LIN {X 0,Y 525.083,Z 545.384,A -85,B 0,C 180,E1 -4788.258,E2 -4788.258} C_VEL
LIN {X 0,Y 525.597,Z 520.306,A -85,B 0,C 180,E1 -4791.163,E2 -4791.163} C_VEL
LIN {X 0,Y 526.091,Z 495.739,A -85,B 0,C 180,E1 -4794.044,E2 -4794.044} C_VEL
LIN {X 0,Y 526.597,Z 472.119,A -85,B 0,C 180,E1 -4796.856,E2 -4796.856} C_VEL
LIN {X 0,Y 524.984,Z 463.792,A -85,B 0,C 180,E1 -4797.939,E2 -4797.939} C_VEL
LIN {X 0,Y 524.003,Z 459.339,A -85,B 0,C 180,E1 -4798.569,E2 -4798.569} C_VEL
LIN {X 0,Y 523.92,Z 459.219,A -85,B 0,C 180,E1 -4801.543,E2 -4801.543} C_VEL
LIN {X 0,Y 523.931,Z 459.225,A -85,B 0,C 180,E1 -4804.289,E2 -4804.289} C_VEL
LIN {X 0,Y 523.905,Z 459.219,A -85,B 0,C 180,E1 -4807.131,E2 -4807.131} C_VEL
LIN {X 0,Y 523.965,Z 459.214,A -85,B 0,C 180,E1 -4810.133,E2 -4810.133} C_VEL
LIN {X 0,Y 523.921,Z 459.219,A -85,B 0,C 180,E1 -4813.166,E2 -4813.166} C_VEL
LIN {X 0,Y 523.936,Z 459.213,A -85,B 0,C 180,E1 -4815.771,E2 -4815.771} C_VEL
LIN {X 0,Y 523.939,Z 459.217,A -85,B 0,C 180,E1 -4818.907,E2 -4818.907} C_VEL
LIN {X 0,Y 523.911,Z 459.221,A -85,B 0,C 180,E1 -4821.898,E2 -4821.898} C_VEL
LIN {X 0,Y 523.933,Z 459.217,A -85,B 0,C 180,E1 -4824.908,E2 -4824.908} C_VEL
LIN {X 0,Y 523.936,Z 459.214,A -85,B 0,C 180,E1 -4827.677,E2 -4827.677} C_VEL
LIN {X 0,Y 523.962,Z 459.216,A -85,B 0,C 180,E1 -4830.673,E2 -4830.673} C_VEL
LIN {X 0,Y 523.97,Z 459.207,A -85,B 0,C 180,E1 -4833.728,E2 -4833.728} C_VEL
LIN {X 0,Y 523.928,Z 459.224,A -85,B 0,C 180,E1 -4836.27,E2 -4836.27} C_VEL
LIN {X 0,Y 523.938,Z 459.216,A -85,B 0,C 180,E1 -4838.766,E2 -4838.766} C_VEL
LIN {X 0,Y 523.945,Z 459.207,A -85,B 0,C 180,E1 -4841.22,E2 -4841.22} C_VEL
LIN {X 0,Y 523.931,Z 459.215,A -85,B 0,C 180,E1 -4843.639,E2 -4843.639} C_VEL
LIN {X 0,Y 523.931,Z 459.22,A -85,B 0,C 180,E1 -4846.028,E2 -4846.028} C_VEL
LIN {X 0,Y 524.002,Z 459.213,A -85,B 0,C 180,E1 -4848.394,E2 -4848.394} C_VEL
LIN {X 0,Y 523.999,Z 459.208,A -85,B 0,C 180,E1 -4851.516,E2 -4851.516} C_VEL
LIN {X 0,Y 524.09,Z 459.2,A -85,B 0,C 180,E1 -4854.614,E2 -4854.614} C_VEL
LIN {X 0,Y 524.103,Z 459.194,A -85,B 0,C 180,E1 -4857.694,E2 -4857.694} C_VEL
LIN {X 0,Y 524.117,Z 459.197,A -85,B 0,C 180,E1 -4860.768,E2 -4860.768} C_VEL
LIN {X 0,Y 524.067,Z 459.199,A -85,B 0,C 180,E1 -4863.075,E2 -4863.075} C_VEL
LIN {X 0,Y 524.042,Z 459.205,A -85,B 0,C 180,E1 -4866.159,E2 -4866.159} C_VEL
LIN {X 0,Y 523.995,Z 459.205,A -85,B 0,C 180,E1 -4869.262,E2 -4869.262} C_VEL
LIN {X 0,Y 523.998,Z 459.207,A -85,B 0,C 180,E1 -4871.743,E2 -4871.743} C_VEL
LIN {X 0,Y 523.984,Z 459.21,A -85,B 0,C 180,E1 -4875.053,E2 -4875.053} C_VEL
LIN {X 0,Y 523.955,Z 459.213,A -85,B 0,C 180,E1 -4877.969,E2 -4877.969} C_VEL
LIN {X 0,Y 523.964,Z 459.217,A -85,B 0,C 180,E1 -4880.41,E2 -4880.41} C_VEL
LIN {X 0,Y 523.909,Z 459.225,A -85,B 0,C 180,E1 -4882.894,E2 -4882.894} C_VEL
LIN {X 0,Y 523.947,Z 459.216,A -85,B 0,C 180,E1 -4885.419,E2 -4885.419} C_VEL
LIN {X 0,Y 523.963,Z 459.21,A -85,B 0,C 180,E1 -4887.999,E2 -4887.999} C_VEL
LIN {X 0,Y 523.945,Z 459.209,A -85,B 0,C 180,E1 -4890.857,E2 -4890.857} C_VEL
LIN {X 0,Y 523.957,Z 459.212,A -85,B 0,C 180,E1 -4893.736,E2 -4893.736} C_VEL
LIN {X 0,Y 523.917,Z 459.221,A -85,B 0,C 180,E1 -4896.405,E2 -4896.405} C_VEL
LIN {X 0,Y 523.918,Z 459.214,A -85,B 0,C 180,E1 -4899.085,E2 -4899.085} C_VEL
LIN {X 0,Y 523.952,Z 459.211,A -85,B 0,C 180,E1 -4902.119,E2 -4902.119} C_VEL
LIN {X 0,Y 523.953,Z 459.216,A -85,B 0,C 180,E1 -4905.309,E2 -4905.309} C_VEL
LIN {X 0,Y 523.92,Z 459.219,A -85,B 0,C 180,E1 -4906.928,E2 -4906.928} C_VEL
LIN {X 0,Y 523.253,Z 459.298,A -85,B 0,C 180,E1 -4907.569,E2 -4907.569} C_VEL
LIN {X 0,Y 520.407,Z 459.654,A -85,B 0,C 180,E1 -4908.611,E2 -4908.611} C_VEL
LIN {X 0,Y 518.001,Z 459.959,A -85,B 0,C 180,E1 -4909.45,E2 -4909.45} C_VEL
LIN {X 0,Y 516.965,Z 460.085,A -85,B 0,C 180,E1 -4910.098,E2 -4910.098} C_VEL
LIN {X 0,Y 516.879,Z 460.096,A -85,B 0,C 180,E1 -4910.317,E2 -4910.317} C_VEL
LIN {X 0,Y 516.882,Z 460.088,A -85,B 0,C 180,E1 -4913.343,E2 -4913.343} C_VEL
LIN {X 0,Y 516.91,Z 460.075,A -85,B 0,C 180,E1 -4916.122,E2 -4916.122} C_VEL
LIN {X 0,Y 516.892,Z 460.099,A -85,B 0,C 180,E1 -4918.936,E2 -4918.936} C_VEL
LIN {X 0,Y 516.919,Z 460.086,A -85,B 0,C 180,E1 -4921.586,E2 -4921.586} C_VEL
LIN {X 0,Y 516.932,Z 460.086,A -85,B 0,C 180,E1 -4924.212,E2 -4924.212} C_VEL
LIN {X 0,Y 516.867,Z 460.102,A -85,B 0,C 180,E1 -4926.777,E2 -4926.777} C_VEL
LIN {X 0,Y 516.942,Z 460.091,A -85,B 0,C 180,E1 -4929.732,E2 -4929.732} C_VEL
LIN {X 0,Y 516.922,Z 460.066,A -85,B 0,C 180,E1 -4932.596,E2 -4932.596} C_VEL
LIN {X 0,Y 516.972,Z 460.252,A -85,B 0,C 180,E1 -4934.934,E2 -4934.934} C_VEL
LIN {X 0,Y 517.22,Z 461.336,A -85,B 0,C 180,E1 -4935.069,E2 -4935.069} C_VEL
LIN {X 0,Y 519.188,Z 467.428,A -85,B 0,C 180,E1 -4935.228,E2 -4935.228} C_VEL
LIN {X 0,Y 518.873,Z 540.381,A -85,B 0,C 180,E1 -4936.264,E2 -4936.264} C_VEL
LIN {X 0,Y 518.787,Z 553.491,A -85,B 0,C 180,E1 -4936.611,E2 -4936.611} C_VEL
LIN {X 0,Y 518.611,Z 565.176,A -85,B 0,C 180,E1 -4937.065,E2 -4937.065} C_VEL
LIN {X 0,Y 518.456,Z 576.909,A -85,B 0,C 180,E1 -4937.679,E2 -4937.679} C_VEL
LIN {X 0,Y 518.112,Z 588.391,A -85,B 0,C 180,E1 -4938.459,E2 -4938.459} C_VEL
LIN {X 0,Y 517.82,Z 598.74,A -85,B 0,C 180,E1 -4939.344,E2 -4939.344} C_VEL
LIN {X 0,Y 517.541,Z 607.185,A -85,B 0,C 180,E1 -4940.227,E2 -4940.227} C_VEL
LIN {X 0,Y 517.36,Z 614.938,A -85,B 0,C 180,E1 -4941.21,E2 -4941.21} C_VEL
LIN {X 0,Y 517.085,Z 622.633,A -85,B 0,C 180,E1 -4942.405,E2 -4942.405} C_VEL
LIN {X 0,Y 516.937,Z 629.45,A -85,B 0,C 180,E1 -4943.756,E2 -4943.756} C_VEL
LIN {X 0,Y 516.696,Z 634.082,A -85,B 0,C 180,E1 -4944.928,E2 -4944.928} C_VEL
LIN {X 0,Y 516.651,Z 637.608,A -85,B 0,C 180,E1 -4946.1,E2 -4946.1} C_VEL
LIN {X 0,Y 516.59,Z 639.435,A -85,B 0,C 180,E1 -4946.881,E2 -4946.881} C_VEL
LIN {X 0,Y 516.577,Z 640.809,A -85,B 0,C 180,E1 -4947.661,E2 -4947.661} C_VEL
LIN {X 0,Y 516.545,Z 642.388,A -85,B 0,C 180,E1 -4949.22,E2 -4949.22} C_VEL
LIN {X 0,Y 516.533,Z 642.622,A -85,B 0,C 180,E1 -4950,E2 -4950} C_VEL
LIN {X 0,Y 516.544,Z 642.442,A -85,B 0,C 180,E1 -4950.78,E2 -4950.78} C_VEL
LIN {X 0,Y 516.577,Z 640.931,A -85,B 0,C 180,E1 -4952.339,E2 -4952.339} C_VEL
LIN {X 0,Y 516.588,Z 639.612,A -85,B 0,C 180,E1 -4953.119,E2 -4953.119} C_VEL
LIN {X 0,Y 516.707,Z 636.807,A -85,B 0,C 180,E1 -4954.29,E2 -4954.29} C_VEL
LIN {X 0,Y 516.814,Z 633.006,A -85,B 0,C 180,E1 -4955.462,E2 -4955.462} C_VEL
LIN {X 0,Y 516.897,Z 627.894,A -85,B 0,C 180,E1 -4956.683,E2 -4956.683} C_VEL
LIN {X 0,Y 517.088,Z 621.918,A -85,B 0,C 180,E1 -4957.811,E2 -4957.811} C_VEL
LIN {X 0,Y 517.386,Z 614.15,A -85,B 0,C 180,E1 -4958.987,E2 -4958.987} C_VEL
LIN {X 0,Y 517.646,Z 604.487,A -85,B 0,C 180,E1 -4960.166,E2 -4960.166} C_VEL
LIN {X 0,Y 517.964,Z 595.465,A -85,B 0,C 180,E1 -4961.049,E2 -4961.049} C_VEL
LIN {X 0,Y 518.262,Z 584.994,A -85,B 0,C 180,E1 -4961.88,E2 -4961.88} C_VEL
LIN {X 0,Y 518.475,Z 573.353,A -85,B 0,C 180,E1 -4962.615,E2 -4962.615} C_VEL
LIN {X 0,Y 518.637,Z 561.959,A -85,B 0,C 180,E1 -4963.169,E2 -4963.169} C_VEL
LIN {X 0,Y 518.811,Z 549.167,A -85,B 0,C 180,E1 -4963.613,E2 -4963.613} C_VEL
LIN {X 0,Y 518.869,Z 537.032,A -85,B 0,C 180,E1 -4963.886,E2 -4963.886} C_VEL
LIN {X 0,Y 519.114,Z 466.662,A -85,B 0,C 180,E1 -4964.875,E2 -4964.875} C_VEL
LIN {X 0,Y 517.159,Z 461.11,A -85,B 0,C 180,E1 -4965.032,E2 -4965.032} C_VEL
LIN {X 0,Y 516.968,Z 460.206,A -85,B 0,C 180,E1 -4965.174,E2 -4965.174} C_VEL
LIN {X 0,Y 516.928,Z 460.073,A -85,B 0,C 180,E1 -4968.222,E2 -4968.222} C_VEL
LIN {X 0,Y 516.915,Z 460.099,A -85,B 0,C 180,E1 -4970.701,E2 -4970.701} C_VEL
LIN {X 0,Y 516.904,Z 460.093,A -85,B 0,C 180,E1 -4974.072,E2 -4974.072} C_VEL
LIN {X 0,Y 516.925,Z 460.087,A -85,B 0,C 180,E1 -4976.657,E2 -4976.657} C_VEL
LIN {X 0,Y 516.911,Z 460.094,A -85,B 0,C 180,E1 -4979.523,E2 -4979.523} C_VEL
LIN {X 0,Y 516.9,Z 460.093,A -85,B 0,C 180,E1 -4982.543,E2 -4982.543} C_VEL
LIN {X 0,Y 516.877,Z 460.098,A -85,B 0,C 180,E1 -4985.331,E2 -4985.331} C_VEL
LIN {X 0,Y 516.88,Z 460.094,A -85,B 0,C 180,E1 -4987.942,E2 -4987.942} C_VEL
LIN {X 0,Y 516.883,Z 460.1,A -85,B 0,C 180,E1 -4990.741,E2 -4990.741} C_VEL
LIN {X 0,Y 516.902,Z 460.092,A -85,B 0,C 180,E1 -4992.828,E2 -4992.828} C_VEL
LIN {X 0,Y 516.919,Z 460.096,A -85,B 0,C 180,E1 -4995.009,E2 -4995.009} C_VEL
LIN {X 0,Y 516.912,Z 460.089,A -85,B 0,C 180,E1 -4998.397,E2 -4998.397} C_VEL
LIN {X 0,Y 516.877,Z 460.096,A -85,B 0,C 180,E1 -5001.284,E2 -5001.284} C_VEL
LIN {X 0,Y 516.885,Z 460.095,A -85,B 0,C 180,E1 -5004.221,E2 -5004.221} C_VEL
LIN {X 0,Y 516.892,Z 460.097,A -85,B 0,C 180,E1 -5007.053,E2 -5007.053} C_VEL
LIN {X 0,Y 516.895,Z 460.083,A -85,B 0,C 180,E1 -5009.796,E2 -5009.796} C_VEL
LIN {X 0,Y 516.923,Z 460.087,A -85,B 0,C 180,E1 -5012.467,E2 -5012.467} C_VEL
LIN {X 0,Y 516.904,Z 460.099,A -85,B 0,C 180,E1 -5015.071,E2 -5015.071} C_VEL
LIN {X 0,Y 516.878,Z 460.092,A -85,B 0,C 180,E1 -5018.462,E2 -5018.462} C_VEL
LIN {X 0,Y 516.896,Z 460.097,A -85,B 0,C 180,E1 -5020.955,E2 -5020.955} C_VEL
LIN {X 0,Y 516.908,Z 460.095,A -85,B 0,C 180,E1 -5023.41,E2 -5023.41} C_VEL
LIN {X 0,Y 516.896,Z 460.095,A -85,B 0,C 180,E1 -5025.834,E2 -5025.834} C_VEL
LIN {X 0,Y 516.948,Z 460.09,A -85,B 0,C 180,E1 -5029.028,E2 -5029.028} C_VEL
LIN {X 0,Y 516.969,Z 460.082,A -85,B 0,C 180,E1 -5032.187,E2 -5032.187} C_VEL
LIN {X 0,Y 517.023,Z 460.076,A -85,B 0,C 180,E1 -5034.54,E2 -5034.54} C_VEL
LIN {X 0,Y 517.075,Z 460.073,A -85,B 0,C 180,E1 -5037.663,E2 -5037.663} C_VEL
LIN {X 0,Y 517.086,Z 460.069,A -85,B 0,C 180,E1 -5040.779,E2 -5040.779} C_VEL
LIN {X 0,Y 517.008,Z 460.081,A -85,B 0,C 180,E1 -5043.117,E2 -5043.117} C_VEL
LIN {X 0,Y 517.001,Z 460.08,A -85,B 0,C 180,E1 -5046.243,E2 -5046.243} C_VEL
LIN {X 0,Y 516.948,Z 460.093,A -85,B 0,C 180,E1 -5049.389,E2 -5049.389} C_VEL
LIN {X 0,Y 516.947,Z 460.09,A -85,B 0,C 180,E1 -5051.81,E2 -5051.81} C_VEL
LIN {X 0,Y 516.934,Z 460.092,A -85,B 0,C 180,E1 -5055.147,E2 -5055.147} C_VEL
LIN {X 0,Y 516.917,Z 460.082,A -85,B 0,C 180,E1 -5058.223,E2 -5058.223} C_VEL
LIN {X 0,Y 516.904,Z 460.088,A -85,B 0,C 180,E1 -5060.702,E2 -5060.702} C_VEL
LIN {X 0,Y 516.903,Z 460.094,A -85,B 0,C 180,E1 -5064.072,E2 -5064.072} C_VEL
LIN {X 0,Y 516.921,Z 460.083,A -85,B 0,C 180,E1 -5066.658,E2 -5066.658} C_VEL
LIN {X 0,Y 516.917,Z 460.096,A -85,B 0,C 180,E1 -5069.527,E2 -5069.527} C_VEL
LIN {X 0,Y 516.894,Z 460.089,A -85,B 0,C 180,E1 -5072.545,E2 -5072.545} C_VEL
LIN {X 0,Y 516.877,Z 460.098,A -85,B 0,C 180,E1 -5075.333,E2 -5075.333} C_VEL
LIN {X 0,Y 516.875,Z 460.099,A -85,B 0,C 180,E1 -5077.944,E2 -5077.944} C_VEL
LIN {X 0,Y 516.88,Z 460.096,A -85,B 0,C 180,E1 -5080.742,E2 -5080.742} C_VEL
LIN {X 0,Y 516.879,Z 460.09,A -85,B 0,C 180,E1 -5082.832,E2 -5082.832} C_VEL
LIN {X 0,Y 516.918,Z 460.085,A -85,B 0,C 180,E1 -5085.011,E2 -5085.011} C_VEL
LIN {X 0,Y 516.919,Z 460.089,A -85,B 0,C 180,E1 -5088.398,E2 -5088.398} C_VEL
LIN {X 0,Y 516.884,Z 460.097,A -85,B 0,C 180,E1 -5091.285,E2 -5091.285} C_VEL
LIN {X 0,Y 516.885,Z 460.1,A -85,B 0,C 180,E1 -5094.222,E2 -5094.222} C_VEL
LIN {X 0,Y 516.895,Z 460.093,A -85,B 0,C 180,E1 -5097.054,E2 -5097.054} C_VEL
LIN {X 0,Y 516.892,Z 460.082,A -85,B 0,C 180,E1 -5099.797,E2 -5099.797} C_VEL
LIN {X 0,Y 516.955,Z 460.3,A -85,B 0,C 180,E1 -5101.255,E2 -5101.255} C_VEL
LIN {X 0,Y 519.648,Z 472.95,A -85,B 0,C 180,E1 -5102.969,E2 -5102.969} C_VEL
LIN {X 0,Y 519.241,Z 493.076,A -85,B 0,C 180,E1 -5105.405,E2 -5105.405} C_VEL
LIN {X 0,Y 518.715,Z 515.897,A -85,B 0,C 180,E1 -5108.125,E2 -5108.125} C_VEL
LIN {X 0,Y 518.097,Z 544.156,A -85,B 0,C 180,E1 -5111.452,E2 -5111.452} C_VEL
LIN {X 0,Y 517.588,Z 571.268,A -85,B 0,C 180,E1 -5114.594,E2 -5114.594} C_VEL
LIN {X 0,Y 519.083,Z 584.74,A -85,B 0,C 180,E1 -5114.848,E2 -5114.848} C_VEL
LIN {X 0,Y 518.599,Z 681.826,A -85,B 0,C 180,E1 -5116.207,E2 -5116.207} C_VEL
LIN {X 0,Y 518.313,Z 695.176,A -85,B 0,C 180,E1 -5116.548,E2 -5116.548} C_VEL
LIN {X 0,Y 518.074,Z 708.587,A -85,B 0,C 180,E1 -5117.066,E2 -5117.066} C_VEL
LIN {X 0,Y 517.77,Z 720.716,A -85,B 0,C 180,E1 -5117.709,E2 -5117.709} C_VEL
LIN {X 0,Y 517.459,Z 732.937,A -85,B 0,C 180,E1 -5118.543,E2 -5118.543} C_VEL
LIN {X 0,Y 517.153,Z 743.295,A -85,B 0,C 180,E1 -5119.429,E2 -5119.429} C_VEL
LIN {X 0,Y 516.925,Z 752.639,A -85,B 0,C 180,E1 -5120.413,E2 -5120.413} C_VEL
LIN {X 0,Y 516.686,Z 761.755,A -85,B 0,C 180,E1 -5121.592,E2 -5121.592} C_VEL
LIN {X 0,Y 516.51,Z 769.109,A -85,B 0,C 180,E1 -5122.77,E2 -5122.77} C_VEL
LIN {X 0,Y 516.454,Z 775.831,A -85,B 0,C 180,E1 -5124.142,E2 -5124.142} C_VEL
LIN {X 0,Y 516.271,Z 780.26,A -85,B 0,C 180,E1 -5125.315,E2 -5125.315} C_VEL
LIN {X 0,Y 516.372,Z 782.633,A -85,B 0,C 180,E1 -5126.098,E2 -5126.098} C_VEL
LIN {X 0,Y 516.282,Z 784.534,A -85,B 0,C 180,E1 -5126.879,E2 -5126.879} C_VEL
LIN {X 0,Y 516.26,Z 785.967,A -85,B 0,C 180,E1 -5127.659,E2 -5127.659} C_VEL
LIN {X 0,Y 516.16,Z 787.598,A -85,B 0,C 180,E1 -5129.22,E2 -5129.22} C_VEL
LIN {X 0,Y 516.154,Z 787.819,A -85,B 0,C 180,E1 -5130,E2 -5130} C_VEL
LIN {X 0,Y 516.16,Z 787.599,A -85,B 0,C 180,E1 -5130.78,E2 -5130.78} C_VEL
LIN {X 0,Y 516.26,Z 785.97,A -85,B 0,C 180,E1 -5132.341,E2 -5132.341} C_VEL
LIN {X 0,Y 516.282,Z 784.538,A -85,B 0,C 180,E1 -5133.121,E2 -5133.121} C_VEL
LIN {X 0,Y 516.326,Z 781.528,A -85,B 0,C 180,E1 -5134.293,E2 -5134.293} C_VEL
LIN {X 0,Y 516.405,Z 777.459,A -85,B 0,C 180,E1 -5135.467,E2 -5135.467} C_VEL
LIN {X 0,Y 516.465,Z 772.035,A -85,B 0,C 180,E1 -5136.678,E2 -5136.678} C_VEL
LIN {X 0,Y 516.578,Z 765.631,A -85,B 0,C 180,E1 -5137.819,E2 -5137.819} C_VEL
LIN {X 0,Y 516.787,Z 757.439,A -85,B 0,C 180,E1 -5138.997,E2 -5138.997} C_VEL
LIN {X 0,Y 517.02,Z 749.107,A -85,B 0,C 180,E1 -5139.98,E2 -5139.98} C_VEL
LIN {X 0,Y 517.279,Z 738.963,A -85,B 0,C 180,E1 -5140.965,E2 -5140.965} C_VEL
LIN {X 0,Y 517.623,Z 727.627,A -85,B 0,C 180,E1 -5141.844,E2 -5141.844} C_VEL
LIN {X 0,Y 517.909,Z 716.373,A -85,B 0,C 180,E1 -5142.54,E2 -5142.54} C_VEL
LIN {X 0,Y 518.124,Z 705.161,A -85,B 0,C 180,E1 -5143.082,E2 -5143.082} C_VEL
LIN {X 0,Y 518.396,Z 692.021,A -85,B 0,C 180,E1 -5143.549,E2 -5143.549} C_VEL
LIN {X 0,Y 518.614,Z 678.964,A -85,B 0,C 180,E1 -5143.843,E2 -5143.843} C_VEL
LIN {X 0,Y 518.889,Z 582.309,A -85,B 0,C 180,E1 -5145.192,E2 -5145.192} C_VEL
LIN {X 0,Y 517.583,Z 571.294,A -85,B 0,C 180,E1 -5145.404,E2 -5145.404} C_VEL
LIN {X 0,Y 518.094,Z 544.154,A -85,B 0,C 180,E1 -5148.548,E2 -5148.548} C_VEL
LIN {X 0,Y 518.613,Z 519.395,A -85,B 0,C 180,E1 -5151.462,E2 -5151.462} C_VEL
LIN {X 0,Y 519.171,Z 494.831,A -85,B 0,C 180,E1 -5154.385,E2 -5154.385} C_VEL
LIN {X 0,Y 519.673,Z 474.807,A -85,B 0,C 180,E1 -5156.801,E2 -5156.801} C_VEL
LIN {X 0,Y 519.444,Z 471.521,A -85,B 0,C 180,E1 -5157.215,E2 -5157.215} C_VEL
LIN {X 0,Y 516.942,Z 460.215,A -85,B 0,C 180,E1 -5158.773,E2 -5158.773} C_VEL
LIN {X 0,Y 516.888,Z 460.093,A -85,B 0,C 180,E1 -5161.109,E2 -5161.109} C_VEL
LIN {X 0,Y 516.906,Z 460.095,A -85,B 0,C 180,E1 -5163.965,E2 -5163.965} C_VEL
LIN {X 0,Y 516.874,Z 460.097,A -85,B 0,C 180,E1 -5166.745,E2 -5166.745} C_VEL
LIN {X 0,Y 516.9,Z 460.095,A -85,B 0,C 180,E1 -5169.719,E2 -5169.719} C_VEL
LIN {X 0,Y 516.903,Z 460.096,A -85,B 0,C 180,E1 -5172.76,E2 -5172.76} C_VEL
LIN {X 0,Y 516.918,Z 460.085,A -85,B 0,C 180,E1 -5175.009,E2 -5175.009} C_VEL
LIN {X 0,Y 516.912,Z 460.099,A -85,B 0,C 180,E1 -5178.397,E2 -5178.397} C_VEL
LIN {X 0,Y 516.877,Z 460.093,A -85,B 0,C 180,E1 -5181.284,E2 -5181.284} C_VEL
LIN {X 0,Y 516.885,Z 460.103,A -85,B 0,C 180,E1 -5184.221,E2 -5184.221} C_VEL
LIN {X 0,Y 516.892,Z 460.091,A -85,B 0,C 180,E1 -5187.053,E2 -5187.053} C_VEL
LIN {X 0,Y 516.895,Z 460.095,A -85,B 0,C 180,E1 -5189.796,E2 -5189.796} C_VEL
LIN {X 0,Y 516.922,Z 460.09,A -85,B 0,C 180,E1 -5192.467,E2 -5192.467} C_VEL
LIN {X 0,Y 516.904,Z 460.092,A -85,B 0,C 180,E1 -5195.071,E2 -5195.071} C_VEL
LIN {X 0,Y 516.878,Z 460.1,A -85,B 0,C 180,E1 -5198.462,E2 -5198.462} C_VEL
LIN {X 0,Y 516.896,Z 460.086,A -85,B 0,C 180,E1 -5200.955,E2 -5200.955} C_VEL
LIN {X 0,Y 516.908,Z 460.089,A -85,B 0,C 180,E1 -5203.41,E2 -5203.41} C_VEL
LIN {X 0,Y 516.886,Z 460.096,A -85,B 0,C 180,E1 -5205.833,E2 -5205.833} C_VEL
LIN {X 0,Y 516.948,Z 460.085,A -85,B 0,C 180,E1 -5209.028,E2 -5209.028} C_VEL
LIN {X 0,Y 516.969,Z 460.088,A -85,B 0,C 180,E1 -5212.187,E2 -5212.187} C_VEL
LIN {X 0,Y 517.051,Z 460.078,A -85,B 0,C 180,E1 -5214.54,E2 -5214.54} C_VEL
LIN {X 0,Y 517.075,Z 460.069,A -85,B 0,C 180,E1 -5217.663,E2 -5217.663} C_VEL
LIN {X 0,Y 517.087,Z 460.073,A -85,B 0,C 180,E1 -5220.779,E2 -5220.779} C_VEL
LIN {X 0,Y 517.008,Z 460.078,A -85,B 0,C 180,E1 -5223.117,E2 -5223.117} C_VEL
LIN {X 0,Y 517.005,Z 460.082,A -85,B 0,C 180,E1 -5226.243,E2 -5226.243} C_VEL
LIN {X 0,Y 516.949,Z 460.082,A -85,B 0,C 180,E1 -5229.389,E2 -5229.389} C_VEL
LIN {X 0,Y 516.947,Z 460.086,A -85,B 0,C 180,E1 -5231.81,E2 -5231.81} C_VEL
LIN {X 0,Y 516.937,Z 460.087,A -85,B 0,C 180,E1 -5235.148,E2 -5235.148} C_VEL
LIN {X 0,Y 516.917,Z 460.091,A -85,B 0,C 180,E1 -5238.223,E2 -5238.223} C_VEL
LIN {X 0,Y 516.904,Z 460.1,A -85,B 0,C 180,E1 -5240.702,E2 -5240.702} C_VEL
LIN {X 0,Y 516.903,Z 460.092,A -85,B 0,C 180,E1 -5244.073,E2 -5244.073} C_VEL
LIN {X 0,Y 516.921,Z 460.097,A -85,B 0,C 180,E1 -5246.658,E2 -5246.658} C_VEL
LIN {X 0,Y 516.918,Z 460.079,A -85,B 0,C 180,E1 -5249.527,E2 -5249.527} C_VEL
LIN {X 0,Y 516.894,Z 460.088,A -85,B 0,C 180,E1 -5252.545,E2 -5252.545} C_VEL
LIN {X 0,Y 516.878,Z 460.098,A -85,B 0,C 180,E1 -5255.333,E2 -5255.333} C_VEL
LIN {X 0,Y 516.876,Z 460.092,A -85,B 0,C 180,E1 -5257.944,E2 -5257.944} C_VEL
LIN {X 0,Y 516.881,Z 460.089,A -85,B 0,C 180,E1 -5260.742,E2 -5260.742} C_VEL
LIN {X 0,Y 516.88,Z 460.1,A -85,B 0,C 180,E1 -5262.832,E2 -5262.832} C_VEL
LIN {X 0,Y 516.919,Z 460.096,A -85,B 0,C 180,E1 -5265.011,E2 -5265.011} C_VEL
LIN {X 0,Y 516.915,Z 460.087,A -85,B 0,C 180,E1 -5268.399,E2 -5268.399} C_VEL
LIN {X 0,Y 516.879,Z 460.096,A -85,B 0,C 180,E1 -5270.317,E2 -5270.317} C_VEL
LIN {X 0,Y 516.212,Z 460.187,A -85,B 0,C 180,E1 -5270.967,E2 -5270.967} C_VEL
LIN {X 0,Y 513.365,Z 460.534,A -85,B 0,C 180,E1 -5272.023,E2 -5272.023} C_VEL
LIN {X 0,Y 510.956,Z 460.834,A -85,B 0,C 180,E1 -5272.873,E2 -5272.873} C_VEL
LIN {X 0,Y 509.916,Z 460.953,A -85,B 0,C 180,E1 -5273.53,E2 -5273.53} C_VEL
LIN {X 0,Y 509.827,Z 460.962,A -85,B 0,C 180,E1 -5273.752,E2 -5273.752} C_VEL
LIN {X 0,Y 509.861,Z 460.955,A -85,B 0,C 180,E1 -5276.54,E2 -5276.54} C_VEL
LIN {X 0,Y 509.846,Z 460.978,A -85,B 0,C 180,E1 -5279.335,E2 -5279.335} C_VEL
LIN {X 0,Y 509.892,Z 460.958,A -85,B 0,C 180,E1 -5282.055,E2 -5282.055} C_VEL
LIN {X 0,Y 509.877,Z 460.968,A -85,B 0,C 180,E1 -5284.705,E2 -5284.705} C_VEL
LIN {X 0,Y 509.828,Z 460.97,A -85,B 0,C 180,E1 -5287.458,E2 -5287.458} C_VEL
LIN {X 0,Y 509.919,Z 460.966,A -85,B 0,C 180,E1 -5289.845,E2 -5289.845} C_VEL
LIN {X 0,Y 509.883,Z 460.94,A -85,B 0,C 180,E1 -5293.175,E2 -5293.175} C_VEL
LIN {X 0,Y 509.945,Z 461.203,A -85,B 0,C 180,E1 -5294.739,E2 -5294.739} C_VEL
LIN {X 0,Y 510.219,Z 462.286,A -85,B 0,C 180,E1 -5294.86,E2 -5294.86} C_VEL
LIN {X 0,Y 512.352,Z 468.914,A -85,B 0,C 180,E1 -5295.033,E2 -5295.033} C_VEL
LIN {X 0,Y 512.024,Z 541.401,A -85,B 0,C 180,E1 -5296.076,E2 -5296.076} C_VEL
LIN {X 0,Y 511.938,Z 554.5,A -85,B 0,C 180,E1 -5296.428,E2 -5296.428} C_VEL
LIN {X 0,Y 511.761,Z 566.178,A -85,B 0,C 180,E1 -5296.889,E2 -5296.889} C_VEL
LIN {X 0,Y 511.593,Z 577.79,A -85,B 0,C 180,E1 -5297.503,E2 -5297.503} C_VEL
LIN {X 0,Y 511.231,Z 589.386,A -85,B 0,C 180,E1 -5298.301,E2 -5298.301} C_VEL
LIN {X 0,Y 510.914,Z 599.735,A -85,B 0,C 180,E1 -5299.198,E2 -5299.198} C_VEL
LIN {X 0,Y 510.618,Z 608.179,A -85,B 0,C 180,E1 -5300.093,E2 -5300.093} C_VEL
LIN {X 0,Y 510.421,Z 615.93,A -85,B 0,C 180,E1 -5301.089,E2 -5301.089} C_VEL
LIN {X 0,Y 510.121,Z 623.624,A -85,B 0,C 180,E1 -5302.3,E2 -5302.3} C_VEL
LIN {X 0,Y 509.954,Z 630.44,A -85,B 0,C 180,E1 -5303.67,E2 -5303.67} C_VEL
LIN {X 0,Y 509.7,Z 635.072,A -85,B 0,C 180,E1 -5304.858,E2 -5304.858} C_VEL
LIN {X 0,Y 509.637,Z 638.598,A -85,B 0,C 180,E1 -5306.046,E2 -5306.046} C_VEL
LIN {X 0,Y 509.57,Z 640.425,A -85,B 0,C 180,E1 -5306.838,E2 -5306.838} C_VEL
LIN {X 0,Y 509.567,Z 641.797,A -85,B 0,C 180,E1 -5307.629,E2 -5307.629} C_VEL
LIN {X 0,Y 509.532,Z 643.375,A -85,B 0,C 180,E1 -5309.21,E2 -5309.21} C_VEL
LIN {X 0,Y 509.52,Z 643.608,A -85,B 0,C 180,E1 -5310,E2 -5310} C_VEL
LIN {X 0,Y 509.532,Z 643.427,A -85,B 0,C 180,E1 -5310.79,E2 -5310.79} C_VEL
LIN {X 0,Y 509.567,Z 641.917,A -85,B 0,C 180,E1 -5312.371,E2 -5312.371} C_VEL
LIN {X 0,Y 509.567,Z 640.6,A -85,B 0,C 180,E1 -5313.162,E2 -5313.162} C_VEL
LIN {X 0,Y 509.696,Z 637.794,A -85,B 0,C 180,E1 -5314.349,E2 -5314.349} C_VEL
LIN {X 0,Y 509.833,Z 633.99,A -85,B 0,C 180,E1 -5315.537,E2 -5315.537} C_VEL
LIN {X 0,Y 509.916,Z 628.888,A -85,B 0,C 180,E1 -5316.773,E2 -5316.773} C_VEL
LIN {X 0,Y 510.125,Z 622.902,A -85,B 0,C 180,E1 -5317.919,E2 -5317.919} C_VEL
LIN {X 0,Y 510.451,Z 615.133,A -85,B 0,C 180,E1 -5319.11,E2 -5319.11} C_VEL
LIN {X 0,Y 510.732,Z 605.47,A -85,B 0,C 180,E1 -5320.305,E2 -5320.305} C_VEL
LIN {X 0,Y 511.048,Z 596.449,A -85,B 0,C 180,E1 -5321.201,E2 -5321.201} C_VEL
LIN {X 0,Y 511.386,Z 585.973,A -85,B 0,C 180,E1 -5322.042,E2 -5322.042} C_VEL
LIN {X 0,Y 511.618,Z 574.331,A -85,B 0,C 180,E1 -5322.787,E2 -5322.787} C_VEL
LIN {X 0,Y 511.784,Z 562.935,A -85,B 0,C 180,E1 -5323.348,E2 -5323.348} C_VEL
LIN {X 0,Y 511.972,Z 550.134,A -85,B 0,C 180,E1 -5323.798,E2 -5323.798} C_VEL
LIN {X 0,Y 511.99,Z 537.991,A -85,B 0,C 180,E1 -5324.076,E2 -5324.076} C_VEL
LIN {X 0,Y 512.312,Z 468.232,A -85,B 0,C 180,E1 -5325.068,E2 -5325.068} C_VEL
LIN {X 0,Y 510.088,Z 461.873,A -85,B 0,C 180,E1 -5325.255,E2 -5325.255} C_VEL
LIN {X 0,Y 509.9,Z 461.031,A -85,B 0,C 180,E1 -5325.422,E2 -5325.422} C_VEL
LIN {X 0,Y 509.869,Z 460.953,A -85,B 0,C 180,E1 -5328.483,E2 -5328.483} C_VEL
LIN {X 0,Y 509.852,Z 460.974,A -85,B 0,C 180,E1 -5331.001,E2 -5331.001} C_VEL
LIN {X 0,Y 509.865,Z 460.972,A -85,B 0,C 180,E1 -5334.426,E2 -5334.426} C_VEL
LIN {X 0,Y 509.884,Z 460.96,A -85,B 0,C 180,E1 -5337.055,E2 -5337.055} C_VEL
LIN {X 0,Y 509.857,Z 460.971,A -85,B 0,C 180,E1 -5339.75,E2 -5339.75} C_VEL
LIN {X 0,Y 509.876,Z 460.97,A -85,B 0,C 180,E1 -5342.774,E2 -5342.774} C_VEL
LIN {X 0,Y 509.837,Z 460.972,A -85,B 0,C 180,E1 -5345.58,E2 -5345.58} C_VEL
LIN {X 0,Y 509.849,Z 460.97,A -85,B 0,C 180,E1 -5348.337,E2 -5348.337} C_VEL
LIN {X 0,Y 509.856,Z 460.969,A -85,B 0,C 180,E1 -5351.424,E2 -5351.424} C_VEL
LIN {X 0,Y 509.853,Z 460.971,A -85,B 0,C 180,E1 -5354.667,E2 -5354.667} C_VEL
LIN {X 0,Y 509.854,Z 460.968,A -85,B 0,C 180,E1 -5358.102,E2 -5358.102} C_VEL
LIN {X 0,Y 509.842,Z 460.961,A -85,B 0,C 180,E1 -5360.647,E2 -5360.647} C_VEL
LIN {X 0,Y 509.83,Z 460.976,A -85,B 0,C 180,E1 -5363.647,E2 -5363.647} C_VEL
LIN {X 0,Y 509.857,Z 460.969,A -85,B 0,C 180,E1 -5366.539,E2 -5366.539} C_VEL
LIN {X 0,Y 509.844,Z 460.963,A -85,B 0,C 180,E1 -5369.334,E2 -5369.334} C_VEL
LIN {X 0,Y 509.888,Z 460.963,A -85,B 0,C 180,E1 -5372.054,E2 -5372.054} C_VEL
LIN {X 0,Y 509.87,Z 460.97,A -85,B 0,C 180,E1 -5374.703,E2 -5374.703} C_VEL
LIN {X 0,Y 509.848,Z 460.974,A -85,B 0,C 180,E1 -5377.449,E2 -5377.449} C_VEL
LIN {X 0,Y 509.908,Z 460.965,A -85,B 0,C 180,E1 -5379.844,E2 -5379.844} C_VEL
LIN {X 0,Y 509.878,Z 460.972,A -85,B 0,C 180,E1 -5383.174,E2 -5383.174} C_VEL
LIN {X 0,Y 509.864,Z 460.974,A -85,B 0,C 180,E1 -5385.634,E2 -5385.634} C_VEL
LIN {X 0,Y 509.908,Z 460.965,A -85,B 0,C 180,E1 -5388.874,E2 -5388.874} C_VEL
LIN {X 0,Y 509.942,Z 460.958,A -85,B 0,C 180,E1 -5392.078,E2 -5392.078} C_VEL
LIN {X 0,Y 509.975,Z 460.954,A -85,B 0,C 180,E1 -5394.464,E2 -5394.464} C_VEL
LIN {X 0,Y 510.046,Z 460.948,A -85,B 0,C 180,E1 -5397.631,E2 -5397.631} C_VEL
LIN {X 0,Y 510.056,Z 460.945,A -85,B 0,C 180,E1 -5400.789,E2 -5400.789} C_VEL
LIN {X 0,Y 509.95,Z 460.96,A -85,B 0,C 180,E1 -5403.16,E2 -5403.16} C_VEL
LIN {X 0,Y 509.969,Z 460.955,A -85,B 0,C 180,E1 -5406.33,E2 -5406.33} C_VEL
LIN {X 0,Y 509.909,Z 460.963,A -85,B 0,C 180,E1 -5408.72,E2 -5408.72} C_VEL
LIN {X 0,Y 509.895,Z 460.967,A -85,B 0,C 180,E1 -5411.932,E2 -5411.932} C_VEL
LIN {X 0,Y 509.884,Z 460.971,A -85,B 0,C 180,E1 -5415.242,E2 -5415.242} C_VEL
LIN {X 0,Y 509.879,Z 460.96,A -85,B 0,C 180,E1 -5418.001,E2 -5418.001} C_VEL
LIN {X 0,Y 509.842,Z 460.969,A -85,B 0,C 180,E1 -5421.002,E2 -5421.002} C_VEL
LIN {X 0,Y 509.861,Z 460.969,A -85,B 0,C 180,E1 -5424.426,E2 -5424.426} C_VEL
LIN {X 0,Y 509.879,Z 460.961,A -85,B 0,C 180,E1 -5427.056,E2 -5427.056} C_VEL
LIN {X 0,Y 509.873,Z 460.976,A -85,B 0,C 180,E1 -5429.75,E2 -5429.75} C_VEL
LIN {X 0,Y 509.87,Z 460.964,A -85,B 0,C 180,E1 -5432.776,E2 -5432.776} C_VEL
LIN {X 0,Y 509.837,Z 460.979,A -85,B 0,C 180,E1 -5435.582,E2 -5435.582} C_VEL
LIN {X 0,Y 509.845,Z 460.971,A -85,B 0,C 180,E1 -5438.339,E2 -5438.339} C_VEL
LIN {X 0,Y 509.853,Z 460.976,A -85,B 0,C 180,E1 -5441.426,E2 -5441.426} C_VEL
LIN {X 0,Y 509.852,Z 460.964,A -85,B 0,C 180,E1 -5444.669,E2 -5444.669} C_VEL
LIN {X 0,Y 509.878,Z 460.969,A -85,B 0,C 180,E1 -5448.101,E2 -5448.101} C_VEL
LIN {X 0,Y 509.857,Z 460.97,A -85,B 0,C 180,E1 -5450.65,E2 -5450.65} C_VEL
LIN {X 0,Y 509.831,Z 460.975,A -85,B 0,C 180,E1 -5453.648,E2 -5453.648} C_VEL
LIN {X 0,Y 509.859,Z 460.969,A -85,B 0,C 180,E1 -5456.54,E2 -5456.54} C_VEL
LIN {X 0,Y 509.845,Z 460.963,A -85,B 0,C 180,E1 -5459.335,E2 -5459.335} C_VEL
LIN {X 0,Y 509.911,Z 461.173,A -85,B 0,C 180,E1 -5461.046,E2 -5461.046} C_VEL
LIN {X 0,Y 512.765,Z 474.548,A -85,B 0,C 180,E1 -5462.886,E2 -5462.886} C_VEL
LIN {X 0,Y 512.253,Z 495.689,A -85,B 0,C 180,E1 -5465.48,E2 -5465.48} C_VEL
LIN {X 0,Y 511.64,Z 522,A -85,B 0,C 180,E1 -5468.654,E2 -5468.654} C_VEL
LIN {X 0,Y 510.926,Z 549.941,A -85,B 0,C 180,E1 -5471.986,E2 -5471.986} C_VEL
LIN {X 0,Y 510.55,Z 570.314,A -85,B 0,C 180,E1 -5474.379,E2 -5474.379} C_VEL
LIN {X 0,Y 512.196,Z 585.14,A -85,B 0,C 180,E1 -5474.659,E2 -5474.659} C_VEL
LIN {X 0,Y 511.697,Z 680.826,A -85,B 0,C 180,E1 -5476.017,E2 -5476.017} C_VEL
LIN {X 0,Y 511.352,Z 694.169,A -85,B 0,C 180,E1 -5476.362,E2 -5476.362} C_VEL
LIN {X 0,Y 511.141,Z 706.449,A -85,B 0,C 180,E1 -5476.837,E2 -5476.837} C_VEL
LIN {X 0,Y 510.839,Z 718.013,A -85,B 0,C 180,E1 -5477.434,E2 -5477.434} C_VEL
LIN {X 0,Y 510.551,Z 729.311,A -85,B 0,C 180,E1 -5478.185,E2 -5478.185} C_VEL
LIN {X 0,Y 510.196,Z 740.135,A -85,B 0,C 180,E1 -5479.082,E2 -5479.082} C_VEL
LIN {X 0,Y 509.92,Z 749.917,A -85,B 0,C 180,E1 -5480.08,E2 -5480.08} C_VEL
LIN {X 0,Y 509.695,Z 757.953,A -85,B 0,C 180,E1 -5481.076,E2 -5481.076} C_VEL
LIN {X 0,Y 509.505,Z 765.821,A -85,B 0,C 180,E1 -5482.271,E2 -5482.271} C_VEL
LIN {X 0,Y 509.344,Z 773.081,A -85,B 0,C 180,E1 -5483.663,E2 -5483.663} C_VEL
LIN {X 0,Y 509.275,Z 777.923,A -85,B 0,C 180,E1 -5484.854,E2 -5484.854} C_VEL
LIN {X 0,Y 509.33,Z 781.64,A -85,B 0,C 180,E1 -5486.044,E2 -5486.044} C_VEL
LIN {X 0,Y 509.239,Z 783.542,A -85,B 0,C 180,E1 -5486.836,E2 -5486.836} C_VEL
LIN {X 0,Y 509.218,Z 784.976,A -85,B 0,C 180,E1 -5487.627,E2 -5487.627} C_VEL
LIN {X 0,Y 509.126,Z 786.613,A -85,B 0,C 180,E1 -5489.209,E2 -5489.209} C_VEL
LIN {X 0,Y 509.144,Z 786.838,A -85,B 0,C 180,E1 -5490,E2 -5490} C_VEL
LIN {X 0,Y 509.157,Z 785.994,A -85,B 0,C 180,E1 -5491.582,E2 -5491.582} C_VEL
LIN {X 0,Y 509.218,Z 784.979,A -85,B 0,C 180,E1 -5492.373,E2 -5492.373} C_VEL
LIN {X 0,Y 509.239,Z 783.546,A -85,B 0,C 180,E1 -5493.164,E2 -5493.164} C_VEL
LIN {X 0,Y 509.256,Z 780.531,A -85,B 0,C 180,E1 -5494.353,E2 -5494.353} C_VEL
LIN {X 0,Y 509.344,Z 776.461,A -85,B 0,C 180,E1 -5495.543,E2 -5495.543} C_VEL
LIN {X 0,Y 509.401,Z 770.659,A -85,B 0,C 180,E1 -5496.844,E2 -5496.844} C_VEL
LIN {X 0,Y 509.563,Z 763.369,A -85,B 0,C 180,E1 -5498.127,E2 -5498.127} C_VEL
LIN {X 0,Y 509.764,Z 754.914,A -85,B 0,C 180,E1 -5499.322,E2 -5499.322} C_VEL
LIN {X 0,Y 510.027,Z 746.266,A -85,B 0,C 180,E1 -5500.319,E2 -5500.319} C_VEL
LIN {X 0,Y 510.341,Z 735.606,A -85,B 0,C 180,E1 -5501.317,E2 -5501.317} C_VEL
LIN {X 0,Y 510.65,Z 723.81,A -85,B 0,C 180,E1 -5502.204,E2 -5502.204} C_VEL
LIN {X 0,Y 510.943,Z 711.619,A -85,B 0,C 180,E1 -5502.915,E2 -5502.915} C_VEL
LIN {X 0,Y 511.346,Z 699.177,A -85,B 0,C 180,E1 -5503.461,E2 -5503.461} C_VEL
LIN {X 0,Y 511.603,Z 686.427,A -85,B 0,C 180,E1 -5503.859,E2 -5503.859} C_VEL
LIN {X 0,Y 511.771,Z 673.155,A -85,B 0,C 180,E1 -5504.108,E2 -5504.108} C_VEL
LIN {X 0,Y 512.144,Z 583.914,A -85,B 0,C 180,E1 -5505.36,E2 -5505.36} C_VEL
LIN {X 0,Y 510.577,Z 570.378,A -85,B 0,C 180,E1 -5505.617,E2 -5505.617} C_VEL
LIN {X 0,Y 511.077,Z 544.614,A -85,B 0,C 180,E1 -5508.645,E2 -5508.645} C_VEL
LIN {X 0,Y 511.638,Z 520.248,A -85,B 0,C 180,E1 -5511.558,E2 -5511.558} C_VEL
LIN {X 0,Y 512.247,Z 495.687,A -85,B 0,C 180,E1 -5514.52,E2 -5514.52} C_VEL
LIN {X 0,Y 512.776,Z 474.527,A -85,B 0,C 180,E1 -5517.114,E2 -5517.114} C_VEL
LIN {X 0,Y 509.902,Z 461.119,A -85,B 0,C 180,E1 -5518.969,E2 -5518.969} C_VEL
LIN {X 0,Y 509.819,Z 460.976,A -85,B 0,C 180,E1 -5521.589,E2 -5521.589} C_VEL
LIN {X 0,Y 509.845,Z 460.979,A -85,B 0,C 180,E1 -5524.413,E2 -5524.413} C_VEL
LIN {X 0,Y 509.814,Z 460.975,A -85,B 0,C 180,E1 -5527.34,E2 -5527.34} C_VEL
LIN {X 0,Y 509.858,Z 460.97,A -85,B 0,C 180,E1 -5530.379,E2 -5530.379} C_VEL
LIN {X 0,Y 509.836,Z 460.974,A -85,B 0,C 180,E1 -5533.063,E2 -5533.063} C_VEL
LIN {X 0,Y 509.826,Z 460.969,A -85,B 0,C 180,E1 -5535.792,E2 -5535.792} C_VEL
LIN {X 0,Y 509.853,Z 460.976,A -85,B 0,C 180,E1 -5538.574,E2 -5538.574} C_VEL
LIN {X 0,Y 509.846,Z 460.971,A -85,B 0,C 180,E1 -5541.786,E2 -5541.786} C_VEL
LIN {X 0,Y 509.84,Z 460.976,A -85,B 0,C 180,E1 -5544.623,E2 -5544.623} C_VEL
LIN {X 0,Y 509.859,Z 460.966,A -85,B 0,C 180,E1 -5547.481,E2 -5547.481} C_VEL
LIN {X 0,Y 509.874,Z 460.976,A -85,B 0,C 180,E1 -5550.268,E2 -5550.268} C_VEL
LIN {X 0,Y 509.879,Z 460.961,A -85,B 0,C 180,E1 -5552.944,E2 -5552.944} C_VEL
LIN {X 0,Y 509.861,Z 460.969,A -85,B 0,C 180,E1 -5555.574,E2 -5555.574} C_VEL
LIN {X 0,Y 509.842,Z 460.969,A -85,B 0,C 180,E1 -5558.998,E2 -5558.998} C_VEL
LIN {X 0,Y 509.879,Z 460.96,A -85,B 0,C 180,E1 -5561.999,E2 -5561.999} C_VEL
LIN {X 0,Y 509.9,Z 460.969,A -85,B 0,C 180,E1 -5564.818,E2 -5564.818} C_VEL
LIN {X 0,Y 509.895,Z 460.967,A -85,B 0,C 180,E1 -5568.121,E2 -5568.121} C_VEL
LIN {X 0,Y 509.909,Z 460.964,A -85,B 0,C 180,E1 -5571.28,E2 -5571.28} C_VEL
LIN {X 0,Y 509.969,Z 460.955,A -85,B 0,C 180,E1 -5573.67,E2 -5573.67} C_VEL
LIN {X 0,Y 509.95,Z 460.962,A -85,B 0,C 180,E1 -5576.84,E2 -5576.84} C_VEL
LIN {X 0,Y 510.056,Z 460.946,A -85,B 0,C 180,E1 -5579.211,E2 -5579.211} C_VEL
LIN {X 0,Y 510.046,Z 460.949,A -85,B 0,C 180,E1 -5582.369,E2 -5582.369} C_VEL
LIN {X 0,Y 510.001,Z 460.952,A -85,B 0,C 180,E1 -5585.536,E2 -5585.536} C_VEL
LIN {X 0,Y 509.942,Z 460.958,A -85,B 0,C 180,E1 -5587.922,E2 -5587.922} C_VEL
LIN {X 0,Y 509.908,Z 460.966,A -85,B 0,C 180,E1 -5591.126,E2 -5591.126} C_VEL
LIN {X 0,Y 509.864,Z 460.973,A -85,B 0,C 180,E1 -5594.366,E2 -5594.366} C_VEL
LIN {X 0,Y 509.894,Z 460.964,A -85,B 0,C 180,E1 -5597.652,E2 -5597.652} C_VEL
LIN {X 0,Y 509.877,Z 460.971,A -85,B 0,C 180,E1 -5600.402,E2 -5600.402} C_VEL
LIN {X 0,Y 509.828,Z 460.973,A -85,B 0,C 180,E1 -5603.564,E2 -5603.564} C_VEL
LIN {X 0,Y 509.906,Z 460.967,A -85,B 0,C 180,E1 -5606.38,E2 -5606.38} C_VEL
LIN {X 0,Y 509.878,Z 460.964,A -85,B 0,C 180,E1 -5608.844,E2 -5608.844} C_VEL
LIN {X 0,Y 509.819,Z 460.965,A -85,B 0,C 180,E1 -5611.59,E2 -5611.59} C_VEL
LIN {X 0,Y 509.849,Z 460.971,A -85,B 0,C 180,E1 -5614.414,E2 -5614.414} C_VEL
LIN {X 0,Y 509.813,Z 460.975,A -85,B 0,C 180,E1 -5617.341,E2 -5617.341} C_VEL
LIN {X 0,Y 509.833,Z 460.962,A -85,B 0,C 180,E1 -5620.383,E2 -5620.383} C_VEL
LIN {X 0,Y 509.82,Z 460.983,A -85,B 0,C 180,E1 -5623.063,E2 -5623.063} C_VEL
LIN {X 0,Y 509.827,Z 460.971,A -85,B 0,C 180,E1 -5625.793,E2 -5625.793} C_VEL
LIN {X 0,Y 509.856,Z 460.968,A -85,B 0,C 180,E1 -5628.576,E2 -5628.576} C_VEL
LIN {X 0,Y 509.85,Z 460.97,A -85,B 0,C 180,E1 -5631.787,E2 -5631.787} C_VEL
LIN {X 0,Y 509.827,Z 460.962,A -85,B 0,C 180,E1 -5633.752,E2 -5633.752} C_VEL
LIN {X 0,Y 509.162,Z 461.045,A -85,B 0,C 180,E1 -5634.412,E2 -5634.412} C_VEL
LIN {X 0,Y 506.344,Z 461.393,A -85,B 0,C 180,E1 -5635.484,E2 -5635.484} C_VEL
LIN {X 0,Y 503.952,Z 461.693,A -85,B 0,C 180,E1 -5636.347,E2 -5636.347} C_VEL
LIN {X 0,Y 502.904,Z 461.827,A -85,B 0,C 180,E1 -5637.014,E2 -5637.014} C_VEL
LIN {X 0,Y 502.808,Z 461.839,A -85,B 0,C 180,E1 -5637.239,E2 -5637.239} C_VEL
LIN {X 0,Y 502.815,Z 461.849,A -85,B 0,C 180,E1 -5640.066,E2 -5640.066} C_VEL
LIN {X 0,Y 502.833,Z 461.839,A -85,B 0,C 180,E1 -5642.534,E2 -5642.534} C_VEL
LIN {X 0,Y 502.828,Z 461.853,A -85,B 0,C 180,E1 -5645.3,E2 -5645.3} C_VEL
LIN {X 0,Y 502.782,Z 461.846,A -85,B 0,C 180,E1 -5647.827,E2 -5647.827} C_VEL
LIN {X 0,Y 502.828,Z 461.849,A -85,B 0,C 180,E1 -5650.401,E2 -5650.401} C_VEL
LIN {X 0,Y 502.83,Z 461.815,A -85,B 0,C 180,E1 -5652.932,E2 -5652.932} C_VEL
LIN {X 0,Y 502.88,Z 462.052,A -85,B 0,C 180,E1 -5654.508,E2 -5654.508} C_VEL
LIN {X 0,Y 503.1,Z 463.022,A -85,B 0,C 180,E1 -5654.632,E2 -5654.632} C_VEL
LIN {X 0,Y 505.485,Z 469.55,A -85,B 0,C 180,E1 -5654.819,E2 -5654.819} C_VEL
LIN {X 0,Y 505.184,Z 542.416,A -85,B 0,C 180,E1 -5655.884,E2 -5655.884} C_VEL
LIN {X 0,Y 505.093,Z 555.507,A -85,B 0,C 180,E1 -5656.241,E2 -5656.241} C_VEL
LIN {X 0,Y 504.916,Z 567.179,A -85,B 0,C 180,E1 -5656.708,E2 -5656.708} C_VEL
LIN {X 0,Y 504.735,Z 578.787,A -85,B 0,C 180,E1 -5657.331,E2 -5657.331} C_VEL
LIN {X 0,Y 504.35,Z 590.382,A -85,B 0,C 180,E1 -5658.139,E2 -5658.139} C_VEL
LIN {X 0,Y 504.011,Z 600.729,A -85,B 0,C 180,E1 -5659.048,E2 -5659.048} C_VEL
LIN {X 0,Y 503.698,Z 609.172,A -85,B 0,C 180,E1 -5659.956,E2 -5659.956} C_VEL
LIN {X 0,Y 503.483,Z 616.922,A -85,B 0,C 180,E1 -5660.965,E2 -5660.965} C_VEL
LIN {X 0,Y 503.159,Z 624.616,A -85,B 0,C 180,E1 -5662.193,E2 -5662.193} C_VEL
LIN {X 0,Y 502.971,Z 631.431,A -85,B 0,C 180,E1 -5663.582,E2 -5663.582} C_VEL
LIN {X 0,Y 502.704,Z 636.062,A -85,B 0,C 180,E1 -5664.786,E2 -5664.786} C_VEL
LIN {X 0,Y 502.624,Z 639.588,A -85,B 0,C 180,E1 -5665.991,E2 -5665.991} C_VEL
LIN {X 0,Y 502.55,Z 641.414,A -85,B 0,C 180,E1 -5666.793,E2 -5666.793} C_VEL
LIN {X 0,Y 502.556,Z 642.784,A -85,B 0,C 180,E1 -5667.596,E2 -5667.596} C_VEL
LIN {X 0,Y 502.518,Z 644.361,A -85,B 0,C 180,E1 -5669.199,E2 -5669.199} C_VEL
LIN {X 0,Y 502.505,Z 644.594,A -85,B 0,C 180,E1 -5670,E2 -5670} C_VEL
LIN {X 0,Y 502.518,Z 644.413,A -85,B 0,C 180,E1 -5670.801,E2 -5670.801} C_VEL
LIN {X 0,Y 502.555,Z 642.903,A -85,B 0,C 180,E1 -5672.404,E2 -5672.404} C_VEL
LIN {X 0,Y 502.547,Z 641.587,A -85,B 0,C 180,E1 -5673.207,E2 -5673.207} C_VEL
LIN {X 0,Y 502.684,Z 638.781,A -85,B 0,C 180,E1 -5674.41,E2 -5674.41} C_VEL
LIN {X 0,Y 502.85,Z 634.975,A -85,B 0,C 180,E1 -5675.614,E2 -5675.614} C_VEL
LIN {X 0,Y 502.936,Z 629.881,A -85,B 0,C 180,E1 -5676.866,E2 -5676.866} C_VEL
LIN {X 0,Y 503.165,Z 623.887,A -85,B 0,C 180,E1 -5678.029,E2 -5678.029} C_VEL
LIN {X 0,Y 503.518,Z 616.116,A -85,B 0,C 180,E1 -5679.237,E2 -5679.237} C_VEL
LIN {X 0,Y 503.819,Z 606.453,A -85,B 0,C 180,E1 -5680.448,E2 -5680.448} C_VEL
LIN {X 0,Y 504.151,Z 597.431,A -85,B 0,C 180,E1 -5681.356,E2 -5681.356} C_VEL
LIN {X 0,Y 504.516,Z 586.953,A -85,B 0,C 180,E1 -5682.209,E2 -5682.209} C_VEL
LIN {X 0,Y 504.767,Z 575.31,A -85,B 0,C 180,E1 -5682.963,E2 -5682.963} C_VEL
LIN {X 0,Y 504.941,Z 563.913,A -85,B 0,C 180,E1 -5683.532,E2 -5683.532} C_VEL
LIN {X 0,Y 505.13,Z 551.106,A -85,B 0,C 180,E1 -5683.989,E2 -5683.989} C_VEL
LIN {X 0,Y 505.163,Z 537.453,A -85,B 0,C 180,E1 -5684.296,E2 -5684.296} C_VEL
LIN {X 0,Y 505.423,Z 469.486,A -85,B 0,C 180,E1 -5685.274,E2 -5685.274} C_VEL
LIN {X 0,Y 502.988,Z 462.672,A -85,B 0,C 180,E1 -5685.484,E2 -5685.484} C_VEL
LIN {X 0,Y 502.845,Z 461.926,A -85,B 0,C 180,E1 -5685.633,E2 -5685.633} C_VEL
LIN {X 0,Y 502.832,Z 461.832,A -85,B 0,C 180,E1 -5688.751,E2 -5688.751} C_VEL
LIN {X 0,Y 502.785,Z 461.85,A -85,B 0,C 180,E1 -5691.311,E2 -5691.311} C_VEL
LIN {X 0,Y 502.786,Z 461.852,A -85,B 0,C 180,E1 -5693.913,E2 -5693.913} C_VEL
LIN {X 0,Y 502.865,Z 461.837,A -85,B 0,C 180,E1 -5696.565,E2 -5696.565} C_VEL
LIN {X 0,Y 502.824,Z 461.852,A -85,B 0,C 180,E1 -5699.287,E2 -5699.287} C_VEL
LIN {X 0,Y 502.787,Z 461.848,A -85,B 0,C 180,E1 -5702.083,E2 -5702.083} C_VEL
LIN {X 0,Y 502.806,Z 461.857,A -85,B 0,C 180,E1 -5704.964,E2 -5704.964} C_VEL
LIN {X 0,Y 502.792,Z 461.849,A -85,B 0,C 180,E1 -5707.953,E2 -5707.953} C_VEL
LIN {X 0,Y 502.818,Z 461.851,A -85,B 0,C 180,E1 -5711.065,E2 -5711.065} C_VEL
LIN {X 0,Y 502.779,Z 461.854,A -85,B 0,C 180,E1 -5713.375,E2 -5713.375} C_VEL
LIN {X 0,Y 502.786,Z 461.854,A -85,B 0,C 180,E1 -5715.66,E2 -5715.66} C_VEL
LIN {X 0,Y 502.814,Z 461.845,A -85,B 0,C 180,E1 -5719.004,E2 -5719.004} C_VEL
LIN {X 0,Y 502.788,Z 461.847,A -85,B 0,C 180,E1 -5722.045,E2 -5722.045} C_VEL
LIN {X 0,Y 502.804,Z 461.856,A -85,B 0,C 180,E1 -5725.034,E2 -5725.034} C_VEL
LIN {X 0,Y 502.781,Z 461.841,A -85,B 0,C 180,E1 -5727.915,E2 -5727.915} C_VEL
LIN {X 0,Y 502.832,Z 461.834,A -85,B 0,C 180,E1 -5730.713,E2 -5730.713} C_VEL
LIN {X 0,Y 502.873,Z 461.846,A -85,B 0,C 180,E1 -5733.434,E2 -5733.434} C_VEL
LIN {X 0,Y 502.783,Z 461.85,A -85,B 0,C 180,E1 -5736.086,E2 -5736.086} C_VEL
LIN {X 0,Y 502.775,Z 461.85,A -85,B 0,C 180,E1 -5738.688,E2 -5738.688} C_VEL
LIN {X 0,Y 502.822,Z 461.855,A -85,B 0,C 180,E1 -5741.248,E2 -5741.248} C_VEL
LIN {X 0,Y 502.814,Z 461.846,A -85,B 0,C 180,E1 -5743.767,E2 -5743.767} C_VEL
LIN {X 0,Y 502.826,Z 461.846,A -85,B 0,C 180,E1 -5746.254,E2 -5746.254} C_VEL
LIN {X 0,Y 502.872,Z 461.84,A -85,B 0,C 180,E1 -5748.717,E2 -5748.717} C_VEL
LIN {X 0,Y 502.893,Z 461.837,A -85,B 0,C 180,E1 -5751.966,E2 -5751.966} C_VEL
LIN {X 0,Y 502.93,Z 461.832,A -85,B 0,C 180,E1 -5754.386,E2 -5754.386} C_VEL
LIN {X 0,Y 503.016,Z 461.824,A -85,B 0,C 180,E1 -5757.598,E2 -5757.598} C_VEL
LIN {X 0,Y 503.017,Z 461.823,A -85,B 0,C 180,E1 -5760,E2 -5760} C_VEL
LIN {X 0,Y 503.016,Z 461.819,A -85,B 0,C 180,E1 -5762.402,E2 -5762.402} C_VEL
LIN {X 0,Y 502.95,Z 461.836,A -85,B 0,C 180,E1 -5765.613,E2 -5765.613} C_VEL
LIN {X 0,Y 502.893,Z 461.839,A -85,B 0,C 180,E1 -5768.033,E2 -5768.033} C_VEL
LIN {X 0,Y 502.871,Z 461.84,A -85,B 0,C 180,E1 -5771.283,E2 -5771.283} C_VEL
LIN {X 0,Y 502.835,Z 461.845,A -85,B 0,C 180,E1 -5774.571,E2 -5774.571} C_VEL
LIN {X 0,Y 502.853,Z 461.836,A -85,B 0,C 180,E1 -5777.907,E2 -5777.907} C_VEL
LIN {X 0,Y 502.819,Z 461.842,A -85,B 0,C 180,E1 -5780.537,E2 -5780.537} C_VEL
LIN {X 0,Y 502.785,Z 461.853,A -85,B 0,C 180,E1 -5783.041,E2 -5783.041} C_VEL
LIN {X 0,Y 502.833,Z 461.845,A -85,B 0,C 180,E1 -5785.676,E2 -5785.676} C_VEL
LIN {X 0,Y 502.835,Z 461.844,A -85,B 0,C 180,E1 -5788.373,E2 -5788.373} C_VEL
LIN {X 0,Y 502.79,Z 461.857,A -85,B 0,C 180,E1 -5791.5,E2 -5791.5} C_VEL
LIN {X 0,Y 502.801,Z 461.849,A -85,B 0,C 180,E1 -5794.446,E2 -5794.446} C_VEL
LIN {X 0,Y 502.775,Z 461.854,A -85,B 0,C 180,E1 -5797.179,E2 -5797.179} C_VEL
LIN {X 0,Y 502.783,Z 461.857,A -85,B 0,C 180,E1 -5800.016,E2 -5800.016} C_VEL
LIN {X 0,Y 502.797,Z 461.847,A -85,B 0,C 180,E1 -5802.2,E2 -5802.2} C_VEL
LIN {X 0,Y 502.796,Z 461.847,A -85,B 0,C 180,E1 -5805.469,E2 -5805.469} C_VEL
LIN {X 0,Y 502.832,Z 461.85,A -85,B 0,C 180,E1 -5807.866,E2 -5807.866} C_VEL
LIN {X 0,Y 502.807,Z 461.849,A -85,B 0,C 180,E1 -5811.026,E2 -5811.026} C_VEL
LIN {X 0,Y 502.78,Z 461.855,A -85,B 0,C 180,E1 -5814.169,E2 -5814.169} C_VEL
LIN {X 0,Y 502.831,Z 461.845,A -85,B 0,C 180,E1 -5816.994,E2 -5816.994} C_VEL
LIN {X 0,Y 502.814,Z 461.831,A -85,B 0,C 180,E1 -5820.066,E2 -5820.066} C_VEL
LIN {X 0,Y 502.885,Z 462.019,A -85,B 0,C 180,E1 -5820.824,E2 -5820.824} C_VEL
LIN {X 0,Y 505.849,Z 475.916,A -85,B 0,C 180,E1 -5822.771,E2 -5822.771} C_VEL
LIN {X 0,Y 505.394,Z 495.062,A -85,B 0,C 180,E1 -5825.158,E2 -5825.158} C_VEL
LIN {X 0,Y 504.663,Z 522.849,A -85,B 0,C 180,E1 -5828.558,E2 -5828.558} C_VEL
LIN {X 0,Y 503.896,Z 549.559,A -85,B 0,C 180,E1 -5831.793,E2 -5831.793} C_VEL
LIN {X 0,Y 503.54,Z 569.39,A -85,B 0,C 180,E1 -5834.16,E2 -5834.16} C_VEL
LIN {X 0,Y 505.301,Z 586.293,A -85,B 0,C 180,E1 -5834.475,E2 -5834.475} C_VEL
LIN {X 0,Y 504.769,Z 679.822,A -85,B 0,C 180,E1 -5835.821,E2 -5835.821} C_VEL
LIN {X 0,Y 504.449,Z 693.17,A -85,B 0,C 180,E1 -5836.172,E2 -5836.172} C_VEL
LIN {X 0,Y 504.149,Z 706.577,A -85,B 0,C 180,E1 -5836.702,E2 -5836.702} C_VEL
LIN {X 0,Y 503.807,Z 718.789,A -85,B 0,C 180,E1 -5837.368,E2 -5837.368} C_VEL
LIN {X 0,Y 503.452,Z 730.926,A -85,B 0,C 180,E1 -5838.22,E2 -5838.22} C_VEL
LIN {X 0,Y 503.086,Z 741.282,A -85,B 0,C 180,E1 -5839.13,E2 -5839.13} C_VEL
LIN {X 0,Y 502.807,Z 750.625,A -85,B 0,C 180,E1 -5840.141,E2 -5840.141} C_VEL
LIN {X 0,Y 502.573,Z 759.749,A -85,B 0,C 180,E1 -5841.354,E2 -5841.354} C_VEL
LIN {X 0,Y 502.366,Z 767.104,A -85,B 0,C 180,E1 -5842.565,E2 -5842.565} C_VEL
LIN {X 0,Y 502.275,Z 772.081,A -85,B 0,C 180,E1 -5843.573,E2 -5843.573} C_VEL
LIN {X 0,Y 502.236,Z 776.929,A -85,B 0,C 180,E1 -5844.781,E2 -5844.781} C_VEL
LIN {X 0,Y 502.285,Z 780.647,A -85,B 0,C 180,E1 -5845.988,E2 -5845.988} C_VEL
LIN {X 0,Y 502.195,Z 782.55,A -85,B 0,C 180,E1 -5846.791,E2 -5846.791} C_VEL
LIN {X 0,Y 502.176,Z 783.985,A -85,B 0,C 180,E1 -5847.594,E2 -5847.594} C_VEL
LIN {X 0,Y 502.12,Z 785.628,A -85,B 0,C 180,E1 -5849.198,E2 -5849.198} C_VEL
LIN {X 0,Y 502.133,Z 785.852,A -85,B 0,C 180,E1 -5850,E2 -5850} C_VEL
LIN {X 0,Y 502.12,Z 785.628,A -85,B 0,C 180,E1 -5850.802,E2 -5850.802} C_VEL
LIN {X 0,Y 502.176,Z 783.988,A -85,B 0,C 180,E1 -5852.406,E2 -5852.406} C_VEL
LIN {X 0,Y 502.195,Z 782.554,A -85,B 0,C 180,E1 -5853.209,E2 -5853.209} C_VEL
LIN {X 0,Y 502.195,Z 779.536,A -85,B 0,C 180,E1 -5854.414,E2 -5854.414} C_VEL
LIN {X 0,Y 502.285,Z 775.464,A -85,B 0,C 180,E1 -5855.621,E2 -5855.621} C_VEL
LIN {X 0,Y 502.333,Z 769.296,A -85,B 0,C 180,E1 -5857.011,E2 -5857.011} C_VEL
LIN {X 0,Y 502.494,Z 762.365,A -85,B 0,C 180,E1 -5858.242,E2 -5858.242} C_VEL
LIN {X 0,Y 502.713,Z 753.91,A -85,B 0,C 180,E1 -5859.454,E2 -5859.454} C_VEL
LIN {X 0,Y 502.961,Z 745.257,A -85,B 0,C 180,E1 -5860.466,E2 -5860.466} C_VEL
LIN {X 0,Y 503.319,Z 734.599,A -85,B 0,C 180,E1 -5861.477,E2 -5861.477} C_VEL
LIN {X 0,Y 503.682,Z 722.677,A -85,B 0,C 180,E1 -5862.384,E2 -5862.384} C_VEL
LIN {X 0,Y 503.981,Z 710.614,A -85,B 0,C 180,E1 -5863.097,E2 -5863.097} C_VEL
LIN {X 0,Y 504.373,Z 698.169,A -85,B 0,C 180,E1 -5863.651,E2 -5863.651} C_VEL
LIN {X 0,Y 504.687,Z 685.426,A -85,B 0,C 180,E1 -5864.053,E2 -5864.053} C_VEL
LIN {X 0,Y 504.87,Z 672.154,A -85,B 0,C 180,E1 -5864.305,E2 -5864.305} C_VEL
LIN {X 0,Y 505.196,Z 584.007,A -85,B 0,C 180,E1 -5865.561,E2 -5865.561} C_VEL
LIN {X 0,Y 503.518,Z 569.36,A -85,B 0,C 180,E1 -5865.842,E2 -5865.842} C_VEL
LIN {X 0,Y 504.039,Z 545.43,A -85,B 0,C 180,E1 -5868.705,E2 -5868.705} C_VEL
LIN {X 0,Y 504.644,Z 521.097,A -85,B 0,C 180,E1 -5871.657,E2 -5871.657} C_VEL
LIN {X 0,Y 505.331,Z 496.547,A -85,B 0,C 180,E1 -5874.659,E2 -5874.659} C_VEL
LIN {X 0,Y 505.869,Z 475.859,A -85,B 0,C 180,E1 -5877.233,E2 -5877.233} C_VEL
LIN {X 0,Y 502.885,Z 462.017,A -85,B 0,C 180,E1 -5879.176,E2 -5879.176} C_VEL
LIN {X 0,Y 502.782,Z 461.859,A -85,B 0,C 180,E1 -5882.084,E2 -5882.084} C_VEL
LIN {X 0,Y 502.797,Z 461.853,A -85,B 0,C 180,E1 -5884.965,E2 -5884.965} C_VEL
LIN {X 0,Y 502.791,Z 461.855,A -85,B 0,C 180,E1 -5887.953,E2 -5887.953} C_VEL
LIN {X 0,Y 502.824,Z 461.843,A -85,B 0,C 180,E1 -5891.064,E2 -5891.064} C_VEL
LIN {X 0,Y 502.778,Z 461.854,A -85,B 0,C 180,E1 -5893.375,E2 -5893.375} C_VEL
LIN {X 0,Y 502.785,Z 461.846,A -85,B 0,C 180,E1 -5895.66,E2 -5895.66} C_VEL
LIN {X 0,Y 502.814,Z 461.849,A -85,B 0,C 180,E1 -5899.004,E2 -5899.004} C_VEL
LIN {X 0,Y 502.788,Z 461.853,A -85,B 0,C 180,E1 -5902.045,E2 -5902.045} C_VEL
LIN {X 0,Y 502.804,Z 461.848,A -85,B 0,C 180,E1 -5905.034,E2 -5905.034} C_VEL
LIN {X 0,Y 502.781,Z 461.85,A -85,B 0,C 180,E1 -5907.915,E2 -5907.915} C_VEL
LIN {X 0,Y 502.832,Z 461.847,A -85,B 0,C 180,E1 -5910.713,E2 -5910.713} C_VEL
LIN {X 0,Y 502.873,Z 461.832,A -85,B 0,C 180,E1 -5913.434,E2 -5913.434} C_VEL
LIN {X 0,Y 502.783,Z 461.855,A -85,B 0,C 180,E1 -5916.086,E2 -5916.086} C_VEL
LIN {X 0,Y 502.775,Z 461.852,A -85,B 0,C 180,E1 -5918.688,E2 -5918.688} C_VEL
LIN {X 0,Y 502.821,Z 461.836,A -85,B 0,C 180,E1 -5921.248,E2 -5921.248} C_VEL
LIN {X 0,Y 502.814,Z 461.845,A -85,B 0,C 180,E1 -5923.767,E2 -5923.767} C_VEL
LIN {X 0,Y 502.822,Z 461.852,A -85,B 0,C 180,E1 -5926.254,E2 -5926.254} C_VEL
LIN {X 0,Y 502.872,Z 461.841,A -85,B 0,C 180,E1 -5928.717,E2 -5928.717} C_VEL
LIN {X 0,Y 502.893,Z 461.839,A -85,B 0,C 180,E1 -5931.967,E2 -5931.967} C_VEL
LIN {X 0,Y 502.95,Z 461.836,A -85,B 0,C 180,E1 -5934.387,E2 -5934.387} C_VEL
LIN {X 0,Y 503.016,Z 461.821,A -85,B 0,C 180,E1 -5937.598,E2 -5937.598} C_VEL
LIN {X 0,Y 503.017,Z 461.824,A -85,B 0,C 180,E1 -5940,E2 -5940} C_VEL
LIN {X 0,Y 503.016,Z 461.824,A -85,B 0,C 180,E1 -5942.402,E2 -5942.402} C_VEL
LIN {X 0,Y 502.953,Z 461.829,A -85,B 0,C 180,E1 -5945.613,E2 -5945.613} C_VEL
LIN {X 0,Y 502.893,Z 461.837,A -85,B 0,C 180,E1 -5948.034,E2 -5948.034} C_VEL
LIN {X 0,Y 502.872,Z 461.841,A -85,B 0,C 180,E1 -5951.283,E2 -5951.283} C_VEL
LIN {X 0,Y 502.842,Z 461.85,A -85,B 0,C 180,E1 -5954.571,E2 -5954.571} C_VEL
LIN {X 0,Y 502.853,Z 461.841,A -85,B 0,C 180,E1 -5957.907,E2 -5957.907} C_VEL
LIN {X 0,Y 502.82,Z 461.852,A -85,B 0,C 180,E1 -5960.537,E2 -5960.537} C_VEL
LIN {X 0,Y 502.788,Z 461.854,A -85,B 0,C 180,E1 -5963.041,E2 -5963.041} C_VEL
LIN {X 0,Y 502.834,Z 461.845,A -85,B 0,C 180,E1 -5965.676,E2 -5965.676} C_VEL
LIN {X 0,Y 502.835,Z 461.844,A -85,B 0,C 180,E1 -5968.373,E2 -5968.373} C_VEL
LIN {X 0,Y 502.79,Z 461.84,A -85,B 0,C 180,E1 -5971.5,E2 -5971.5} C_VEL
LIN {X 0,Y 502.801,Z 461.85,A -85,B 0,C 180,E1 -5974.446,E2 -5974.446} C_VEL
LIN {X 0,Y 502.775,Z 461.854,A -85,B 0,C 180,E1 -5977.179,E2 -5977.179} C_VEL
LIN {X 0,Y 502.783,Z 461.838,A -85,B 0,C 180,E1 -5980.016,E2 -5980.016} C_VEL
LIN {X 0,Y 502.798,Z 461.846,A -85,B 0,C 180,E1 -5982.2,E2 -5982.2} C_VEL
LIN {X 0,Y 502.797,Z 461.849,A -85,B 0,C 180,E1 -5985.469,E2 -5985.469} C_VEL
LIN {X 0,Y 502.827,Z 461.84,A -85,B 0,C 180,E1 -5987.865,E2 -5987.865} C_VEL
LIN {X 0,Y 502.801,Z 461.856,A -85,B 0,C 180,E1 -5991.025,E2 -5991.025} C_VEL
LIN {X 0,Y 502.781,Z 461.838,A -85,B 0,C 180,E1 -5994.169,E2 -5994.169} C_VEL
LIN {X 0,Y 502.808,Z 461.839,A -85,B 0,C 180,E1 -5997.239,E2 -5997.239} C_VEL
LIN {X 0,Y 502.108,Z 461.935,A -85,B 0,C 180,E1 -5997.908,E2 -5997.908} C_VEL
LIN {X 0,Y 499.243,Z 462.299,A -85,B 0,C 180,E1 -5998.994,E2 -5998.994} C_VEL
LIN {X 0,Y 496.847,Z 462.594,A -85,B 0,C 180,E1 -5999.869,E2 -5999.869} C_VEL
LIN {X 0,Y 495.831,Z 462.721,A -85,B 0,C 180,E1 -6000.544,E2 -6000.544} C_VEL
LIN {X 0,Y 495.753,Z 462.726,A -85,B 0,C 180,E1 -6000.773,E2 -6000.773} C_VEL
LIN {X 0,Y 495.792,Z 462.719,A -85,B 0,C 180,E1 -6003.933,E2 -6003.933} C_VEL
LIN {X 0,Y 495.761,Z 462.723,A -85,B 0,C 180,E1 -6007.14,E2 -6007.14} C_VEL
LIN {X 0,Y 495.78,Z 462.726,A -85,B 0,C 180,E1 -6010.111,E2 -6010.111} C_VEL
LIN {X 0,Y 495.782,Z 462.691,A -85,B 0,C 180,E1 -6012.682,E2 -6012.682} C_VEL
LIN {X 0,Y 495.841,Z 462.896,A -85,B 0,C 180,E1 -6014.272,E2 -6014.272} C_VEL
LIN {X 0,Y 496.024,Z 463.713,A -85,B 0,C 180,E1 -6014.396,E2 -6014.396} C_VEL
LIN {X 0,Y 498.606,Z 470.885,A -85,B 0,C 180,E1 -6014.609,E2 -6014.609} C_VEL
LIN {X 0,Y 498.348,Z 543.429,A -85,B 0,C 180,E1 -6015.686,E2 -6015.686} C_VEL
LIN {X 0,Y 498.256,Z 556.511,A -85,B 0,C 180,E1 -6016.048,E2 -6016.048} C_VEL
LIN {X 0,Y 498.075,Z 568.178,A -85,B 0,C 180,E1 -6016.522,E2 -6016.522} C_VEL
LIN {X 0,Y 497.877,Z 580.182,A -85,B 0,C 180,E1 -6017.179,E2 -6017.179} C_VEL
LIN {X 0,Y 497.472,Z 591.376,A -85,B 0,C 180,E1 -6017.973,E2 -6017.973} C_VEL
LIN {X 0,Y 497.112,Z 601.723,A -85,B 0,C 180,E1 -6018.894,E2 -6018.894} C_VEL
LIN {X 0,Y 496.782,Z 610.164,A -85,B 0,C 180,E1 -6019.815,E2 -6019.815} C_VEL
LIN {X 0,Y 496.546,Z 617.913,A -85,B 0,C 180,E1 -6020.838,E2 -6020.838} C_VEL
LIN {X 0,Y 496.198,Z 625.606,A -85,B 0,C 180,E1 -6022.083,E2 -6022.083} C_VEL
LIN {X 0,Y 495.996,Z 631.365,A -85,B 0,C 180,E1 -6023.245,E2 -6023.245} C_VEL
LIN {X 0,Y 495.875,Z 635.646,A -85,B 0,C 180,E1 -6024.306,E2 -6024.306} C_VEL
LIN {X 0,Y 495.677,Z 639.534,A -85,B 0,C 180,E1 -6025.528,E2 -6025.528} C_VEL
LIN {X 0,Y 495.531,Z 642.404,A -85,B 0,C 180,E1 -6026.748,E2 -6026.748} C_VEL
LIN {X 0,Y 495.543,Z 643.772,A -85,B 0,C 180,E1 -6027.562,E2 -6027.562} C_VEL
LIN {X 0,Y 495.503,Z 645.348,A -85,B 0,C 180,E1 -6029.187,E2 -6029.187} C_VEL
LIN {X 0,Y 495.489,Z 645.581,A -85,B 0,C 180,E1 -6030,E2 -6030} C_VEL
LIN {X 0,Y 495.503,Z 645.399,A -85,B 0,C 180,E1 -6030.813,E2 -6030.813} C_VEL
LIN {X 0,Y 495.542,Z 643.889,A -85,B 0,C 180,E1 -6032.438,E2 -6032.438} C_VEL
LIN {X 0,Y 495.527,Z 642.575,A -85,B 0,C 180,E1 -6033.252,E2 -6033.252} C_VEL
LIN {X 0,Y 495.674,Z 639.768,A -85,B 0,C 180,E1 -6034.473,E2 -6034.473} C_VEL
LIN {X 0,Y 495.866,Z 635.96,A -85,B 0,C 180,E1 -6035.694,E2 -6035.694} C_VEL
LIN {X 0,Y 495.958,Z 630.871,A -85,B 0,C 180,E1 -6036.962,E2 -6036.962} C_VEL
LIN {X 0,Y 496.207,Z 624.872,A -85,B 0,C 180,E1 -6038.142,E2 -6038.142} C_VEL
LIN {X 0,Y 496.586,Z 617.1,A -85,B 0,C 180,E1 -6039.367,E2 -6039.367} C_VEL
LIN {X 0,Y 496.908,Z 607.437,A -85,B 0,C 180,E1 -6040.595,E2 -6040.595} C_VEL
LIN {X 0,Y 497.26,Z 598.414,A -85,B 0,C 180,E1 -6041.515,E2 -6041.515} C_VEL
LIN {X 0,Y 497.649,Z 587.934,A -85,B 0,C 180,E1 -6042.38,E2 -6042.38} C_VEL
LIN {X 0,Y 497.904,Z 576.446,A -85,B 0,C 180,E1 -6043.136,E2 -6043.136} C_VEL
LIN {X 0,Y 498.098,Z 565.224,A -85,B 0,C 180,E1 -6043.707,E2 -6043.707} C_VEL
LIN {X 0,Y 498.301,Z 552.079,A -85,B 0,C 180,E1 -6044.185,E2 -6044.185} C_VEL
LIN {X 0,Y 498.322,Z 539.915,A -85,B 0,C 180,E1 -6044.471,E2 -6044.471} C_VEL
LIN {X 0,Y 498.6,Z 471.031,A -85,B 0,C 180,E1 -6045.48,E2 -6045.48} C_VEL
LIN {X 0,Y 495.963,Z 463.582,A -85,B 0,C 180,E1 -6045.707,E2 -6045.707} C_VEL
LIN {X 0,Y 495.804,Z 462.806,A -85,B 0,C 180,E1 -6045.861,E2 -6045.861} C_VEL
LIN {X 0,Y 495.787,Z 462.713,A -85,B 0,C 180,E1 -6049.028,E2 -6049.028} C_VEL
LIN {X 0,Y 495.744,Z 462.724,A -85,B 0,C 180,E1 -6051.628,E2 -6051.628} C_VEL
LIN {X 0,Y 495.779,Z 462.732,A -85,B 0,C 180,E1 -6054.872,E2 -6054.872} C_VEL
LIN {X 0,Y 495.814,Z 462.711,A -85,B 0,C 180,E1 -6056.974,E2 -6056.974} C_VEL
LIN {X 0,Y 495.765,Z 462.727,A -85,B 0,C 180,E1 -6060.146,E2 -6060.146} C_VEL
LIN {X 0,Y 495.792,Z 462.728,A -85,B 0,C 180,E1 -6063.244,E2 -6063.244} C_VEL
LIN {X 0,Y 495.724,Z 462.728,A -85,B 0,C 180,E1 -6066.089,E2 -6066.089} C_VEL
LIN {X 0,Y 495.762,Z 462.729,A -85,B 0,C 180,E1 -6068.768,E2 -6068.768} C_VEL
LIN {X 0,Y 495.774,Z 462.719,A -85,B 0,C 180,E1 -6071.778,E2 -6071.778} C_VEL
LIN {X 0,Y 495.745,Z 462.735,A -85,B 0,C 180,E1 -6075.139,E2 -6075.139} C_VEL
LIN {X 0,Y 495.753,Z 462.724,A -85,B 0,C 180,E1 -6078.218,E2 -6078.218} C_VEL
LIN {X 0,Y 495.746,Z 462.729,A -85,B 0,C 180,E1 -6081.408,E2 -6081.408} C_VEL
LIN {X 0,Y 495.752,Z 462.728,A -85,B 0,C 180,E1 -6084.462,E2 -6084.462} C_VEL
LIN {X 0,Y 495.763,Z 462.72,A -85,B 0,C 180,E1 -6087.405,E2 -6087.405} C_VEL
LIN {X 0,Y 495.774,Z 462.71,A -85,B 0,C 180,E1 -6090.254,E2 -6090.254} C_VEL
LIN {X 0,Y 495.826,Z 462.723,A -85,B 0,C 180,E1 -6093.248,E2 -6093.248} C_VEL
LIN {X 0,Y 495.744,Z 462.729,A -85,B 0,C 180,E1 -6095.724,E2 -6095.724} C_VEL
LIN {X 0,Y 495.739,Z 462.725,A -85,B 0,C 180,E1 -6098.371,E2 -6098.371} C_VEL
LIN {X 0,Y 495.776,Z 462.728,A -85,B 0,C 180,E1 -6100.971,E2 -6100.971} C_VEL
LIN {X 0,Y 495.772,Z 462.725,A -85,B 0,C 180,E1 -6103.53,E2 -6103.53} C_VEL
LIN {X 0,Y 495.789,Z 462.723,A -85,B 0,C 180,E1 -6106.055,E2 -6106.055} C_VEL
LIN {X 0,Y 495.845,Z 462.715,A -85,B 0,C 180,E1 -6108.555,E2 -6108.555} C_VEL
LIN {X 0,Y 495.864,Z 462.714,A -85,B 0,C 180,E1 -6111.852,E2 -6111.852} C_VEL
LIN {X 0,Y 495.888,Z 462.709,A -85,B 0,C 180,E1 -6114.306,E2 -6114.306} C_VEL
LIN {X 0,Y 495.985,Z 462.699,A -85,B 0,C 180,E1 -6117.564,E2 -6117.564} C_VEL
LIN {X 0,Y 495.988,Z 462.698,A -85,B 0,C 180,E1 -6120,E2 -6120} C_VEL
LIN {X 0,Y 495.985,Z 462.695,A -85,B 0,C 180,E1 -6122.436,E2 -6122.436} C_VEL
LIN {X 0,Y 495.904,Z 462.713,A -85,B 0,C 180,E1 -6125.693,E2 -6125.693} C_VEL
LIN {X 0,Y 495.864,Z 462.714,A -85,B 0,C 180,E1 -6128.148,E2 -6128.148} C_VEL
LIN {X 0,Y 495.845,Z 462.716,A -85,B 0,C 180,E1 -6131.445,E2 -6131.445} C_VEL
LIN {X 0,Y 495.78,Z 462.724,A -85,B 0,C 180,E1 -6134.783,E2 -6134.783} C_VEL
LIN {X 0,Y 495.779,Z 462.726,A -85,B 0,C 180,E1 -6137.319,E2 -6137.319} C_VEL
LIN {X 0,Y 495.77,Z 462.725,A -85,B 0,C 180,E1 -6139.89,E2 -6139.89} C_VEL
LIN {X 0,Y 495.752,Z 462.728,A -85,B 0,C 180,E1 -6142.862,E2 -6142.862} C_VEL
LIN {X 0,Y 495.791,Z 462.716,A -85,B 0,C 180,E1 -6146.068,E2 -6146.068} C_VEL
LIN {X 0,Y 495.773,Z 462.723,A -85,B 0,C 180,E1 -6148.815,E2 -6148.815} C_VEL
LIN {X 0,Y 495.752,Z 462.731,A -85,B 0,C 180,E1 -6151.727,E2 -6151.727} C_VEL
LIN {X 0,Y 495.771,Z 462.724,A -85,B 0,C 180,E1 -6154.696,E2 -6154.696} C_VEL
LIN {X 0,Y 495.726,Z 462.736,A -85,B 0,C 180,E1 -6157.562,E2 -6157.562} C_VEL
LIN {X 0,Y 495.761,Z 462.727,A -85,B 0,C 180,E1 -6160.701,E2 -6160.701} C_VEL
LIN {X 0,Y 495.729,Z 462.723,A -85,B 0,C 180,E1 -6164.002,E2 -6164.002} C_VEL
LIN {X 0,Y 495.759,Z 462.729,A -85,B 0,C 180,E1 -6167.122,E2 -6167.122} C_VEL
LIN {X 0,Y 495.78,Z 462.726,A -85,B 0,C 180,E1 -6170.365,E2 -6170.365} C_VEL
LIN {X 0,Y 495.73,Z 462.731,A -85,B 0,C 180,E1 -6173.457,E2 -6173.457} C_VEL
LIN {X 0,Y 495.759,Z 462.726,A -85,B 0,C 180,E1 -6176.437,E2 -6176.437} C_VEL
LIN {X 0,Y 495.752,Z 462.715,A -85,B 0,C 180,E1 -6179.314,E2 -6179.314} C_VEL
LIN {X 0,Y 495.861,Z 462.976,A -85,B 0,C 180,E1 -6180.625,E2 -6180.625} C_VEL
LIN {X 0,Y 498.986,Z 477.847,A -85,B 0,C 180,E1 -6182.728,E2 -6182.728} C_VEL
LIN {X 0,Y 498.32,Z 499.162,A -85,B 0,C 180,E1 -6185.415,E2 -6185.415} C_VEL
LIN {X 0,Y 497.674,Z 523.694,A -85,B 0,C 180,E1 -6188.46,E2 -6188.46} C_VEL
LIN {X 0,Y 496.88,Z 550.338,A -85,B 0,C 180,E1 -6191.737,E2 -6191.737} C_VEL
LIN {X 0,Y 496.515,Z 568.465,A -85,B 0,C 180,E1 -6193.935,E2 -6193.935} C_VEL
LIN {X 0,Y 498.429,Z 586.852,A -85,B 0,C 180,E1 -6194.279,E2 -6194.279} C_VEL
LIN {X 0,Y 497.876,Z 678.822,A -85,B 0,C 180,E1 -6195.62,E2 -6195.62} C_VEL
LIN {X 0,Y 497.578,Z 692.175,A -85,B 0,C 180,E1 -6195.977,E2 -6195.977} C_VEL
LIN {X 0,Y 497.191,Z 705.571,A -85,B 0,C 180,E1 -6196.513,E2 -6196.513} C_VEL
LIN {X 0,Y 496.853,Z 717.117,A -85,B 0,C 180,E1 -6197.145,E2 -6197.145} C_VEL
LIN {X 0,Y 496.495,Z 728.608,A -85,B 0,C 180,E1 -6197.949,E2 -6197.949} C_VEL
LIN {X 0,Y 496.083,Z 739.207,A -85,B 0,C 180,E1 -6198.871,E2 -6198.871} C_VEL
LIN {X 0,Y 495.798,Z 747.9,A -85,B 0,C 180,E1 -6199.794,E2 -6199.794} C_VEL
LIN {X 0,Y 495.545,Z 755.938,A -85,B 0,C 180,E1 -6200.819,E2 -6200.819} C_VEL
LIN {X 0,Y 495.365,Z 763.814,A -85,B 0,C 180,E1 -6202.049,E2 -6202.049} C_VEL
LIN {X 0,Y 495.203,Z 771.08,A -85,B 0,C 180,E1 -6203.481,E2 -6203.481} C_VEL
LIN {X 0,Y 495.196,Z 775.935,A -85,B 0,C 180,E1 -6204.707,E2 -6204.707} C_VEL
LIN {X 0,Y 495.22,Z 779.652,A -85,B 0,C 180,E1 -6205.931,E2 -6205.931} C_VEL
LIN {X 0,Y 495.151,Z 781.558,A -85,B 0,C 180,E1 -6206.745,E2 -6206.745} C_VEL
LIN {X 0,Y 495.134,Z 782.994,A -85,B 0,C 180,E1 -6207.56,E2 -6207.56} C_VEL
LIN {X 0,Y 495.112,Z 784.642,A -85,B 0,C 180,E1 -6209.187,E2 -6209.187} C_VEL
LIN {X 0,Y 495.121,Z 784.866,A -85,B 0,C 180,E1 -6210,E2 -6210} C_VEL
LIN {X 0,Y 495.112,Z 784.643,A -85,B 0,C 180,E1 -6210.813,E2 -6210.813} C_VEL
LIN {X 0,Y 495.134,Z 782.997,A -85,B 0,C 180,E1 -6212.44,E2 -6212.44} C_VEL
LIN {X 0,Y 495.151,Z 781.562,A -85,B 0,C 180,E1 -6213.255,E2 -6213.255} C_VEL
LIN {X 0,Y 495.141,Z 778.541,A -85,B 0,C 180,E1 -6214.477,E2 -6214.477} C_VEL
LIN {X 0,Y 495.265,Z 773.265,A -85,B 0,C 180,E1 -6216.003,E2 -6216.003} C_VEL
LIN {X 0,Y 495.276,Z 767.155,A -85,B 0,C 180,E1 -6217.337,E2 -6217.337} C_VEL
LIN {X 0,Y 495.477,Z 760.1,A -85,B 0,C 180,E1 -6218.565,E2 -6218.565} C_VEL
LIN {X 0,Y 495.679,Z 751.278,A -85,B 0,C 180,E1 -6219.796,E2 -6219.796} C_VEL
LIN {X 0,Y 495.975,Z 742.265,A -85,B 0,C 180,E1 -6220.821,E2 -6220.821} C_VEL
LIN {X 0,Y 496.404,Z 731.206,A -85,B 0,C 180,E1 -6221.846,E2 -6221.846} C_VEL
LIN {X 0,Y 496.741,Z 720.635,A -85,B 0,C 180,E1 -6222.63,E2 -6222.63} C_VEL
LIN {X 0,Y 497.07,Z 708.607,A -85,B 0,C 180,E1 -6223.334,E2 -6223.334} C_VEL
LIN {X 0,Y 497.493,Z 695.858,A -85,B 0,C 180,E1 -6223.895,E2 -6223.895} C_VEL
LIN {X 0,Y 497.816,Z 683.4,A -85,B 0,C 180,E1 -6224.277,E2 -6224.277} C_VEL
LIN {X 0,Y 498.012,Z 667.565,A -85,B 0,C 180,E1 -6224.558,E2 -6224.558} C_VEL
LIN {X 0,Y 498.373,Z 585.023,A -85,B 0,C 180,E1 -6225.75,E2 -6225.75} C_VEL
LIN {X 0,Y 496.492,Z 568.273,A -85,B 0,C 180,E1 -6226.079,E2 -6226.079} C_VEL
LIN {X 0,Y 497.113,Z 542.78,A -85,B 0,C 180,E1 -6229.189,E2 -6229.189} C_VEL
LIN {X 0,Y 497.846,Z 516.696,A -85,B 0,C 180,E1 -6232.405,E2 -6232.405} C_VEL
LIN {X 0,Y 498.526,Z 493.324,A -85,B 0,C 180,E1 -6235.314,E2 -6235.314} C_VEL
LIN {X 0,Y 498.989,Z 477.783,A -85,B 0,C 180,E1 -6237.279,E2 -6237.279} C_VEL
LIN {X 0,Y 495.861,Z 462.975,A -85,B 0,C 180,E1 -6239.375,E2 -6239.375} C_VEL
LIN {X 0,Y 495.764,Z 462.708,A -85,B 0,C 180,E1 -6240.146,E2 -6240.146} C_VEL
LIN {X 0,Y 495.791,Z 462.722,A -85,B 0,C 180,E1 -6243.244,E2 -6243.244} C_VEL
LIN {X 0,Y 495.717,Z 462.733,A -85,B 0,C 180,E1 -6246.088,E2 -6246.088} C_VEL
LIN {X 0,Y 495.766,Z 462.727,A -85,B 0,C 180,E1 -6248.768,E2 -6248.768} C_VEL
LIN {X 0,Y 495.779,Z 462.724,A -85,B 0,C 180,E1 -6251.778,E2 -6251.778} C_VEL
LIN {X 0,Y 495.745,Z 462.721,A -85,B 0,C 180,E1 -6255.139,E2 -6255.139} C_VEL
LIN {X 0,Y 495.752,Z 462.73,A -85,B 0,C 180,E1 -6258.218,E2 -6258.218} C_VEL
LIN {X 0,Y 495.745,Z 462.725,A -85,B 0,C 180,E1 -6261.408,E2 -6261.408} C_VEL
LIN {X 0,Y 495.752,Z 462.733,A -85,B 0,C 180,E1 -6264.462,E2 -6264.462} C_VEL
LIN {X 0,Y 495.763,Z 462.721,A -85,B 0,C 180,E1 -6267.405,E2 -6267.405} C_VEL
LIN {X 0,Y 495.775,Z 462.732,A -85,B 0,C 180,E1 -6270.254,E2 -6270.254} C_VEL
LIN {X 0,Y 495.826,Z 462.71,A -85,B 0,C 180,E1 -6273.248,E2 -6273.248} C_VEL
LIN {X 0,Y 495.744,Z 462.728,A -85,B 0,C 180,E1 -6275.724,E2 -6275.724} C_VEL
LIN {X 0,Y 495.734,Z 462.735,A -85,B 0,C 180,E1 -6278.371,E2 -6278.371} C_VEL
LIN {X 0,Y 495.776,Z 462.715,A -85,B 0,C 180,E1 -6280.971,E2 -6280.971} C_VEL
LIN {X 0,Y 495.771,Z 462.722,A -85,B 0,C 180,E1 -6283.53,E2 -6283.53} C_VEL
LIN {X 0,Y 495.784,Z 462.726,A -85,B 0,C 180,E1 -6286.055,E2 -6286.055} C_VEL
LIN {X 0,Y 495.845,Z 462.717,A -85,B 0,C 180,E1 -6288.555,E2 -6288.555} C_VEL
LIN {X 0,Y 495.864,Z 462.714,A -85,B 0,C 180,E1 -6291.852,E2 -6291.852} C_VEL
LIN {X 0,Y 495.904,Z 462.713,A -85,B 0,C 180,E1 -6294.307,E2 -6294.307} C_VEL
LIN {X 0,Y 495.985,Z 462.697,A -85,B 0,C 180,E1 -6297.564,E2 -6297.564} C_VEL
LIN {X 0,Y 495.988,Z 462.699,A -85,B 0,C 180,E1 -6300,E2 -6300} C_VEL
LIN {X 0,Y 495.985,Z 462.7,A -85,B 0,C 180,E1 -6302.436,E2 -6302.436} C_VEL
LIN {X 0,Y 495.907,Z 462.707,A -85,B 0,C 180,E1 -6305.693,E2 -6305.693} C_VEL
LIN {X 0,Y 495.864,Z 462.713,A -85,B 0,C 180,E1 -6308.148,E2 -6308.148} C_VEL
LIN {X 0,Y 495.845,Z 462.715,A -85,B 0,C 180,E1 -6311.445,E2 -6311.445} C_VEL
LIN {X 0,Y 495.785,Z 462.726,A -85,B 0,C 180,E1 -6314.783,E2 -6314.783} C_VEL
LIN {X 0,Y 495.779,Z 462.724,A -85,B 0,C 180,E1 -6317.319,E2 -6317.319} C_VEL
LIN {X 0,Y 495.769,Z 462.725,A -85,B 0,C 180,E1 -6319.891,E2 -6319.891} C_VEL
LIN {X 0,Y 495.749,Z 462.731,A -85,B 0,C 180,E1 -6322.861,E2 -6322.861} C_VEL
LIN {X 0,Y 495.791,Z 462.723,A -85,B 0,C 180,E1 -6326.068,E2 -6326.068} C_VEL
LIN {X 0,Y 495.773,Z 462.72,A -85,B 0,C 180,E1 -6328.815,E2 -6328.815} C_VEL
LIN {X 0,Y 495.752,Z 462.715,A -85,B 0,C 180,E1 -6331.727,E2 -6331.727} C_VEL
LIN {X 0,Y 495.771,Z 462.729,A -85,B 0,C 180,E1 -6334.696,E2 -6334.696} C_VEL
LIN {X 0,Y 495.726,Z 462.728,A -85,B 0,C 180,E1 -6337.562,E2 -6337.562} C_VEL
LIN {X 0,Y 495.762,Z 462.717,A -85,B 0,C 180,E1 -6340.701,E2 -6340.701} C_VEL
LIN {X 0,Y 495.73,Z 462.73,A -85,B 0,C 180,E1 -6344.002,E2 -6344.002} C_VEL
LIN {X 0,Y 495.731,Z 462.727,A -85,B 0,C 180,E1 -6347.119,E2 -6347.119} C_VEL
LIN {X 0,Y 495.757,Z 462.727,A -85,B 0,C 180,E1 -6349.954,E2 -6349.954} C_VEL
LIN {X 0,Y 495.729,Z 462.731,A -85,B 0,C 180,E1 -6352.554,E2 -6352.554} C_VEL
LIN {X 0,Y 495.782,Z 462.702,A -85,B 0,C 180,E1 -6355.458,E2 -6355.458} C_VEL
LIN {X 0,Y 495.758,Z 462.725,A -85,B 0,C 180,E1 -6358.365,E2 -6358.365} C_VEL
LIN {X 0,Y 495.753,Z 462.726,A -85,B 0,C 180,E1 -6360.773,E2 -6360.773} C_VEL
LIN {X 0,Y 495.097,Z 462.806,A -85,B 0,C 180,E1 -6361.452,E2 -6361.452} C_VEL
LIN {X 0,Y 492.24,Z 463.157,A -85,B 0,C 180,E1 -6362.554,E2 -6362.554} C_VEL
LIN {X 0,Y 489.831,Z 463.457,A -85,B 0,C 180,E1 -6363.443,E2 -6363.443} C_VEL
LIN {X 0,Y 488.816,Z 463.588,A -85,B 0,C 180,E1 -6364.129,E2 -6364.129} C_VEL
LIN {X 0,Y 488.744,Z 463.597,A -85,B 0,C 180,E1 -6364.362,E2 -6364.362} C_VEL
LIN {X 0,Y 488.724,Z 463.599,A -85,B 0,C 180,E1 -6367.154,E2 -6367.154} C_VEL
LIN {X 0,Y 488.731,Z 463.606,A -85,B 0,C 180,E1 -6369.811,E2 -6369.811} C_VEL
LIN {X 0,Y 488.731,Z 463.569,A -85,B 0,C 180,E1 -6372.424,E2 -6372.424} C_VEL
LIN {X 0,Y 488.791,Z 463.782,A -85,B 0,C 180,E1 -6374.039,E2 -6374.039} C_VEL
LIN {X 0,Y 489.015,Z 464.828,A -85,B 0,C 180,E1 -6374.175,E2 -6374.175} C_VEL
LIN {X 0,Y 491.868,Z 472.627,A -85,B 0,C 180,E1 -6374.404,E2 -6374.404} C_VEL
LIN {X 0,Y 491.518,Z 544.44,A -85,B 0,C 180,E1 -6375.483,E2 -6375.483} C_VEL
LIN {X 0,Y 491.426,Z 557.514,A -85,B 0,C 180,E1 -6375.85,E2 -6375.85} C_VEL
LIN {X 0,Y 491.258,Z 569.517,A -85,B 0,C 180,E1 -6376.347,E2 -6376.347} C_VEL
LIN {X 0,Y 491.03,Z 580.774,A -85,B 0,C 180,E1 -6376.971,E2 -6376.971} C_VEL
LIN {X 0,Y 490.599,Z 592.37,A -85,B 0,C 180,E1 -6377.802,E2 -6377.802} C_VEL
LIN {X 0,Y 490.217,Z 602.716,A -85,B 0,C 180,E1 -6378.736,E2 -6378.736} C_VEL
LIN {X 0,Y 489.869,Z 611.155,A -85,B 0,C 180,E1 -6379.669,E2 -6379.669} C_VEL
LIN {X 0,Y 489.61,Z 618.904,A -85,B 0,C 180,E1 -6380.707,E2 -6380.707} C_VEL
LIN {X 0,Y 489.239,Z 626.597,A -85,B 0,C 180,E1 -6381.97,E2 -6381.97} C_VEL
LIN {X 0,Y 489.018,Z 632.356,A -85,B 0,C 180,E1 -6383.148,E2 -6383.148} C_VEL
LIN {X 0,Y 488.891,Z 636.635,A -85,B 0,C 180,E1 -6384.225,E2 -6384.225} C_VEL
LIN {X 0,Y 488.668,Z 640.524,A -85,B 0,C 180,E1 -6385.463,E2 -6385.463} C_VEL
LIN {X 0,Y 488.512,Z 643.394,A -85,B 0,C 180,E1 -6386.701,E2 -6386.701} C_VEL
LIN {X 0,Y 488.529,Z 644.759,A -85,B 0,C 180,E1 -6387.527,E2 -6387.527} C_VEL
LIN {X 0,Y 488.419,Z 645.745,A -85,B 0,C 180,E1 -6388.351,E2 -6388.351} C_VEL
LIN {X 0,Y 488.487,Z 646.335,A -85,B 0,C 180,E1 -6389.176,E2 -6389.176} C_VEL
LIN {X 0,Y 488.472,Z 646.568,A -85,B 0,C 180,E1 -6390,E2 -6390} C_VEL
LIN {X 0,Y 488.487,Z 646.386,A -85,B 0,C 180,E1 -6390.824,E2 -6390.824} C_VEL
LIN {X 0,Y 488.419,Z 645.829,A -85,B 0,C 180,E1 -6391.649,E2 -6391.649} C_VEL
LIN {X 0,Y 488.528,Z 644.876,A -85,B 0,C 180,E1 -6392.473,E2 -6392.473} C_VEL
LIN {X 0,Y 488.507,Z 643.563,A -85,B 0,C 180,E1 -6393.299,E2 -6393.299} C_VEL
LIN {X 0,Y 488.664,Z 640.756,A -85,B 0,C 180,E1 -6394.537,E2 -6394.537} C_VEL
LIN {X 0,Y 488.882,Z 636.945,A -85,B 0,C 180,E1 -6395.775,E2 -6395.775} C_VEL
LIN {X 0,Y 488.982,Z 631.861,A -85,B 0,C 180,E1 -6397.061,E2 -6397.061} C_VEL
LIN {X 0,Y 489.252,Z 625.857,A -85,B 0,C 180,E1 -6398.259,E2 -6398.259} C_VEL
LIN {X 0,Y 489.656,Z 618.085,A -85,B 0,C 180,E1 -6399.5,E2 -6399.5} C_VEL
LIN {X 0,Y 490,Z 608.421,A -85,B 0,C 180,E1 -6400.746,E2 -6400.746} C_VEL
LIN {X 0,Y 490.374,Z 599.397,A -85,B 0,C 180,E1 -6401.679,E2 -6401.679} C_VEL
LIN {X 0,Y 490.787,Z 588.916,A -85,B 0,C 180,E1 -6402.556,E2 -6402.556} C_VEL
LIN {X 0,Y 491.063,Z 577.427,A -85,B 0,C 180,E1 -6403.322,E2 -6403.322} C_VEL
LIN {X 0,Y 491.266,Z 566.203,A -85,B 0,C 180,E1 -6403.901,E2 -6403.901} C_VEL
LIN {X 0,Y 491.47,Z 553.054,A -85,B 0,C 180,E1 -6404.386,E2 -6404.386} C_VEL
LIN {X 0,Y 491.505,Z 539.382,A -85,B 0,C 180,E1 -6404.702,E2 -6404.702} C_VEL
LIN {X 0,Y 491.8,Z 472.493,A -85,B 0,C 180,E1 -6405.692,E2 -6405.692} C_VEL
LIN {X 0,Y 488.91,Z 464.41,A -85,B 0,C 180,E1 -6405.946,E2 -6405.946} C_VEL
LIN {X 0,Y 488.765,Z 463.685,A -85,B 0,C 180,E1 -6406.095,E2 -6406.095} C_VEL
LIN {X 0,Y 488.748,Z 463.595,A -85,B 0,C 180,E1 -6409.313,E2 -6409.313} C_VEL
LIN {X 0,Y 488.7,Z 463.599,A -85,B 0,C 180,E1 -6411.956,E2 -6411.956} C_VEL
LIN {X 0,Y 488.745,Z 463.605,A -85,B 0,C 180,E1 -6415.052,E2 -6415.052} C_VEL
LIN {X 0,Y 488.746,Z 463.59,A -85,B 0,C 180,E1 -6417.396,E2 -6417.396} C_VEL
LIN {X 0,Y 488.71,Z 463.607,A -85,B 0,C 180,E1 -6420.362,E2 -6420.362} C_VEL
LIN {X 0,Y 488.734,Z 463.605,A -85,B 0,C 180,E1 -6423.484,E2 -6423.484} C_VEL
LIN {X 0,Y 488.685,Z 463.606,A -85,B 0,C 180,E1 -6426.355,E2 -6426.355} C_VEL
LIN {X 0,Y 488.699,Z 463.613,A -85,B 0,C 180,E1 -6429.253,E2 -6429.253} C_VEL
LIN {X 0,Y 488.72,Z 463.599,A -85,B 0,C 180,E1 -6431.601,E2 -6431.601} C_VEL
LIN {X 0,Y 488.708,Z 463.606,A -85,B 0,C 180,E1 -6434.801,E2 -6434.801} C_VEL
LIN {X 0,Y 488.687,Z 463.608,A -85,B 0,C 180,E1 -6437.474,E2 -6437.474} C_VEL
LIN {X 0,Y 488.728,Z 463.588,A -85,B 0,C 180,E1 -6439.676,E2 -6439.676} C_VEL
LIN {X 0,Y 488.677,Z 463.609,A -85,B 0,C 180,E1 -6442.841,E2 -6442.841} C_VEL
LIN {X 0,Y 488.729,Z 463.6,A -85,B 0,C 180,E1 -6445.887,E2 -6445.887} C_VEL
LIN {X 0,Y 488.69,Z 463.596,A -85,B 0,C 180,E1 -6448.82,E2 -6448.82} C_VEL
LIN {X 0,Y 488.74,Z 463.599,A -85,B 0,C 180,E1 -6451.671,E2 -6451.671} C_VEL
LIN {X 0,Y 488.743,Z 463.601,A -85,B 0,C 180,E1 -6454.444,E2 -6454.444} C_VEL
LIN {X 0,Y 488.712,Z 463.607,A -85,B 0,C 180,E1 -6457.153,E2 -6457.153} C_VEL
LIN {X 0,Y 488.72,Z 463.605,A -85,B 0,C 180,E1 -6459.81,E2 -6459.81} C_VEL
LIN {X 0,Y 488.726,Z 463.601,A -85,B 0,C 180,E1 -6462.423,E2 -6462.423} C_VEL
LIN {X 0,Y 488.755,Z 463.598,A -85,B 0,C 180,E1 -6464.999,E2 -6464.999} C_VEL
LIN {X 0,Y 488.798,Z 463.592,A -85,B 0,C 180,E1 -6468.387,E2 -6468.387} C_VEL
LIN {X 0,Y 488.809,Z 463.594,A -85,B 0,C 180,E1 -6471.733,E2 -6471.733} C_VEL
LIN {X 0,Y 488.847,Z 463.587,A -85,B 0,C 180,E1 -6474.224,E2 -6474.224} C_VEL
LIN {X 0,Y 488.952,Z 463.574,A -85,B 0,C 180,E1 -6477.529,E2 -6477.529} C_VEL
LIN {X 0,Y 488.959,Z 463.574,A -85,B 0,C 180,E1 -6480,E2 -6480} C_VEL
LIN {X 0,Y 488.952,Z 463.571,A -85,B 0,C 180,E1 -6482.471,E2 -6482.471} C_VEL
LIN {X 0,Y 488.86,Z 463.589,A -85,B 0,C 180,E1 -6485.776,E2 -6485.776} C_VEL
LIN {X 0,Y 488.809,Z 463.592,A -85,B 0,C 180,E1 -6488.267,E2 -6488.267} C_VEL
LIN {X 0,Y 488.798,Z 463.596,A -85,B 0,C 180,E1 -6491.613,E2 -6491.613} C_VEL
LIN {X 0,Y 488.752,Z 463.601,A -85,B 0,C 180,E1 -6495.001,E2 -6495.001} C_VEL
LIN {X 0,Y 488.746,Z 463.587,A -85,B 0,C 180,E1 -6498.443,E2 -6498.443} C_VEL
LIN {X 0,Y 488.698,Z 463.603,A -85,B 0,C 180,E1 -6501.071,E2 -6501.071} C_VEL
LIN {X 0,Y 488.684,Z 463.613,A -85,B 0,C 180,E1 -6503.746,E2 -6503.746} C_VEL
LIN {X 0,Y 488.791,Z 463.586,A -85,B 0,C 180,E1 -6506.946,E2 -6506.946} C_VEL
LIN {X 0,Y 488.712,Z 463.605,A -85,B 0,C 180,E1 -6510.365,E2 -6510.365} C_VEL
LIN {X 0,Y 488.729,Z 463.601,A -85,B 0,C 180,E1 -6513.485,E2 -6513.485} C_VEL
LIN {X 0,Y 488.683,Z 463.609,A -85,B 0,C 180,E1 -6516.356,E2 -6516.356} C_VEL
LIN {X 0,Y 488.696,Z 463.606,A -85,B 0,C 180,E1 -6519.255,E2 -6519.255} C_VEL
LIN {X 0,Y 488.703,Z 463.611,A -85,B 0,C 180,E1 -6521.601,E2 -6521.601} C_VEL
LIN {X 0,Y 488.707,Z 463.597,A -85,B 0,C 180,E1 -6524.802,E2 -6524.802} C_VEL
LIN {X 0,Y 488.728,Z 463.608,A -85,B 0,C 180,E1 -6527.48,E2 -6527.48} C_VEL
LIN {X 0,Y 488.74,Z 463.601,A -85,B 0,C 180,E1 -6530.751,E2 -6530.751} C_VEL
LIN {X 0,Y 488.681,Z 463.608,A -85,B 0,C 180,E1 -6533.869,E2 -6533.869} C_VEL
LIN {X 0,Y 488.737,Z 463.6,A -85,B 0,C 180,E1 -6536.878,E2 -6536.878} C_VEL
LIN {X 0,Y 488.791,Z 463.785,A -85,B 0,C 180,E1 -6540.38,E2 -6540.38} C_VEL
LIN {X 0,Y 492.006,Z 478.691,A -85,B 0,C 180,E1 -6542.536,E2 -6542.536} C_VEL
LIN {X 0,Y 491.723,Z 491.71,A -85,B 0,C 180,E1 -6544.216,E2 -6544.216} C_VEL
LIN {X 0,Y 490.933,Z 514.027,A -85,B 0,C 180,E1 -6547.04,E2 -6547.04} C_VEL
LIN {X 0,Y 490.293,Z 534.947,A -85,B 0,C 180,E1 -6549.66,E2 -6549.66} C_VEL
LIN {X 0,Y 489.674,Z 559.058,A -85,B 0,C 180,E1 -6552.674,E2 -6552.674} C_VEL
LIN {X 0,Y 489.498,Z 567.294,A -85,B 0,C 180,E1 -6553.688,E2 -6553.688} C_VEL
LIN {X 0,Y 491.563,Z 586.912,A -85,B 0,C 180,E1 -6554.069,E2 -6554.069} C_VEL
LIN {X 0,Y 490.983,Z 677.82,A -85,B 0,C 180,E1 -6555.414,E2 -6555.414} C_VEL
LIN {X 0,Y 490.649,Z 691.17,A -85,B 0,C 180,E1 -6555.775,E2 -6555.775} C_VEL
LIN {X 0,Y 490.273,Z 704.57,A -85,B 0,C 180,E1 -6556.319,E2 -6556.319} C_VEL
LIN {X 0,Y 489.86,Z 716.166,A -85,B 0,C 180,E1 -6556.962,E2 -6556.962} C_VEL
LIN {X 0,Y 489.504,Z 727.603,A -85,B 0,C 180,E1 -6557.774,E2 -6557.774} C_VEL
LIN {X 0,Y 488.997,Z 738.191,A -85,B 0,C 180,E1 -6558.708,E2 -6558.708} C_VEL
LIN {X 0,Y 488.75,Z 746.893,A -85,B 0,C 180,E1 -6559.645,E2 -6559.645} C_VEL
LIN {X 0,Y 488.493,Z 754.934,A -85,B 0,C 180,E1 -6560.686,E2 -6560.686} C_VEL
LIN {X 0,Y 488.32,Z 762.814,A -85,B 0,C 180,E1 -6561.934,E2 -6561.934} C_VEL
LIN {X 0,Y 488.142,Z 770.08,A -85,B 0,C 180,E1 -6563.386,E2 -6563.386} C_VEL
LIN {X 0,Y 488.134,Z 774.938,A -85,B 0,C 180,E1 -6564.63,E2 -6564.63} C_VEL
LIN {X 0,Y 488.145,Z 778.654,A -85,B 0,C 180,E1 -6565.872,E2 -6565.872} C_VEL
LIN {X 0,Y 488.105,Z 780.566,A -85,B 0,C 180,E1 -6566.698,E2 -6566.698} C_VEL
LIN {X 0,Y 488.091,Z 782.003,A -85,B 0,C 180,E1 -6567.524,E2 -6567.524} C_VEL
LIN {X 0,Y 488.102,Z 783.656,A -85,B 0,C 180,E1 -6569.175,E2 -6569.175} C_VEL
LIN {X 0,Y 488.107,Z 783.88,A -85,B 0,C 180,E1 -6570,E2 -6570} C_VEL
LIN {X 0,Y 488.102,Z 783.657,A -85,B 0,C 180,E1 -6570.825,E2 -6570.825} C_VEL
LIN {X 0,Y 488.091,Z 782.006,A -85,B 0,C 180,E1 -6572.476,E2 -6572.476} C_VEL
LIN {X 0,Y 488.105,Z 780.57,A -85,B 0,C 180,E1 -6573.302,E2 -6573.302} C_VEL
LIN {X 0,Y 488.091,Z 777.547,A -85,B 0,C 180,E1 -6574.542,E2 -6574.542} C_VEL
LIN {X 0,Y 488.203,Z 772.439,A -85,B 0,C 180,E1 -6576.048,E2 -6576.048} C_VEL
LIN {X 0,Y 488.236,Z 766.157,A -85,B 0,C 180,E1 -6577.444,E2 -6577.444} C_VEL
LIN {X 0,Y 488.39,Z 759.093,A -85,B 0,C 180,E1 -6578.69,E2 -6578.69} C_VEL
LIN {X 0,Y 488.632,Z 750.272,A -85,B 0,C 180,E1 -6579.939,E2 -6579.939} C_VEL
LIN {X 0,Y 488.955,Z 741.259,A -85,B 0,C 180,E1 -6580.979,E2 -6580.979} C_VEL
LIN {X 0,Y 489.357,Z 731.396,A -85,B 0,C 180,E1 -6581.914,E2 -6581.914} C_VEL
LIN {X 0,Y 489.701,Z 720.767,A -85,B 0,C 180,E1 -6582.736,E2 -6582.736} C_VEL
LIN {X 0,Y 490.084,Z 708.607,A -85,B 0,C 180,E1 -6583.475,E2 -6583.475} C_VEL
LIN {X 0,Y 490.543,Z 696.166,A -85,B 0,C 180,E1 -6584.043,E2 -6584.043} C_VEL
LIN {X 0,Y 490.89,Z 683.424,A -85,B 0,C 180,E1 -6584.456,E2 -6584.456} C_VEL
LIN {X 0,Y 491.114,Z 670.157,A -85,B 0,C 180,E1 -6584.714,E2 -6584.714} C_VEL
LIN {X 0,Y 491.432,Z 585.021,A -85,B 0,C 180,E1 -6585.963,E2 -6585.963} C_VEL
LIN {X 0,Y 489.48,Z 567.471,A -85,B 0,C 180,E1 -6586.302,E2 -6586.302} C_VEL
LIN {X 0,Y 490.116,Z 541.862,A -85,B 0,C 180,E1 -6589.474,E2 -6589.474} C_VEL
LIN {X 0,Y 490.864,Z 517.528,A -85,B 0,C 180,E1 -6592.519,E2 -6592.519} C_VEL
LIN {X 0,Y 491.615,Z 493.735,A -85,B 0,C 180,E1 -6595.526,E2 -6595.526} C_VEL
LIN {X 0,Y 492.044,Z 478.667,A -85,B 0,C 180,E1 -6597.464,E2 -6597.464} C_VEL
LIN {X 0,Y 488.775,Z 463.735,A -85,B 0,C 180,E1 -6599.636,E2 -6599.636} C_VEL
LIN {X 0,Y 488.736,Z 463.6,A -85,B 0,C 180,E1 -6603.122,E2 -6603.122} C_VEL
LIN {X 0,Y 488.675,Z 463.609,A -85,B 0,C 180,E1 -6606.131,E2 -6606.131} C_VEL
LIN {X 0,Y 488.74,Z 463.6,A -85,B 0,C 180,E1 -6609.249,E2 -6609.249} C_VEL
LIN {X 0,Y 488.728,Z 463.609,A -85,B 0,C 180,E1 -6612.52,E2 -6612.52} C_VEL
LIN {X 0,Y 488.707,Z 463.597,A -85,B 0,C 180,E1 -6615.198,E2 -6615.198} C_VEL
LIN {X 0,Y 488.703,Z 463.611,A -85,B 0,C 180,E1 -6618.399,E2 -6618.399} C_VEL
LIN {X 0,Y 488.699,Z 463.604,A -85,B 0,C 180,E1 -6620.946,E2 -6620.946} C_VEL
LIN {X 0,Y 488.679,Z 463.611,A -85,B 0,C 180,E1 -6623.868,E2 -6623.868} C_VEL
LIN {X 0,Y 488.733,Z 463.599,A -85,B 0,C 180,E1 -6626.877,E2 -6626.877} C_VEL
LIN {X 0,Y 488.727,Z 463.605,A -85,B 0,C 180,E1 -6629.781,E2 -6629.781} C_VEL
LIN {X 0,Y 488.791,Z 463.586,A -85,B 0,C 180,E1 -6633.054,E2 -6633.054} C_VEL
LIN {X 0,Y 488.684,Z 463.613,A -85,B 0,C 180,E1 -6636.254,E2 -6636.254} C_VEL
LIN {X 0,Y 488.737,Z 463.596,A -85,B 0,C 180,E1 -6639.175,E2 -6639.175} C_VEL
LIN {X 0,Y 488.75,Z 463.588,A -85,B 0,C 180,E1 -6641.627,E2 -6641.627} C_VEL
LIN {X 0,Y 488.752,Z 463.601,A -85,B 0,C 180,E1 -6644.999,E2 -6644.999} C_VEL
LIN {X 0,Y 488.798,Z 463.596,A -85,B 0,C 180,E1 -6648.387,E2 -6648.387} C_VEL
LIN {X 0,Y 488.809,Z 463.592,A -85,B 0,C 180,E1 -6651.733,E2 -6651.733} C_VEL
LIN {X 0,Y 488.861,Z 463.589,A -85,B 0,C 180,E1 -6654.224,E2 -6654.224} C_VEL
LIN {X 0,Y 488.952,Z 463.573,A -85,B 0,C 180,E1 -6657.529,E2 -6657.529} C_VEL
LIN {X 0,Y 488.959,Z 463.575,A -85,B 0,C 180,E1 -6660,E2 -6660} C_VEL
LIN {X 0,Y 488.952,Z 463.575,A -85,B 0,C 180,E1 -6662.471,E2 -6662.471} C_VEL
LIN {X 0,Y 488.863,Z 463.585,A -85,B 0,C 180,E1 -6665.776,E2 -6665.776} C_VEL
LIN {X 0,Y 488.809,Z 463.593,A -85,B 0,C 180,E1 -6668.267,E2 -6668.267} C_VEL
LIN {X 0,Y 488.798,Z 463.592,A -85,B 0,C 180,E1 -6671.613,E2 -6671.613} C_VEL
LIN {X 0,Y 488.755,Z 463.598,A -85,B 0,C 180,E1 -6675.001,E2 -6675.001} C_VEL
LIN {X 0,Y 488.746,Z 463.603,A -85,B 0,C 180,E1 -6678.443,E2 -6678.443} C_VEL
LIN {X 0,Y 488.699,Z 463.606,A -85,B 0,C 180,E1 -6681.071,E2 -6681.071} C_VEL
LIN {X 0,Y 488.685,Z 463.606,A -85,B 0,C 180,E1 -6683.746,E2 -6683.746} C_VEL
LIN {X 0,Y 488.791,Z 463.597,A -85,B 0,C 180,E1 -6686.946,E2 -6686.946} C_VEL
LIN {X 0,Y 488.712,Z 463.592,A -85,B 0,C 180,E1 -6690.366,E2 -6690.366} C_VEL
LIN {X 0,Y 488.73,Z 463.601,A -85,B 0,C 180,E1 -6693.485,E2 -6693.485} C_VEL
LIN {X 0,Y 488.683,Z 463.61,A -85,B 0,C 180,E1 -6696.356,E2 -6696.356} C_VEL
LIN {X 0,Y 488.696,Z 463.595,A -85,B 0,C 180,E1 -6699.255,E2 -6699.255} C_VEL
LIN {X 0,Y 488.704,Z 463.602,A -85,B 0,C 180,E1 -6701.601,E2 -6701.601} C_VEL
LIN {X 0,Y 488.708,Z 463.612,A -85,B 0,C 180,E1 -6704.802,E2 -6704.802} C_VEL
LIN {X 0,Y 488.692,Z 463.602,A -85,B 0,C 180,E1 -6707.476,E2 -6707.476} C_VEL
LIN {X 0,Y 488.73,Z 463.603,A -85,B 0,C 180,E1 -6709.677,E2 -6709.677} C_VEL
LIN {X 0,Y 488.68,Z 463.606,A -85,B 0,C 180,E1 -6712.842,E2 -6712.842} C_VEL
LIN {X 0,Y 488.733,Z 463.581,A -85,B 0,C 180,E1 -6715.888,E2 -6715.888} C_VEL
LIN {X 0,Y 488.694,Z 463.61,A -85,B 0,C 180,E1 -6718.821,E2 -6718.821} C_VEL
LIN {X 0,Y 488.745,Z 463.593,A -85,B 0,C 180,E1 -6721.672,E2 -6721.672} C_VEL
LIN {X 0,Y 488.744,Z 463.597,A -85,B 0,C 180,E1 -6724.362,E2 -6724.362} C_VEL
LIN {X 0,Y 488.1,Z 463.687,A -85,B 0,C 180,E1 -6725.05,E2 -6725.05} C_VEL
LIN {X 0,Y 485.23,Z 464.039,A -85,B 0,C 180,E1 -6726.166,E2 -6726.166} C_VEL
LIN {X 0,Y 482.782,Z 464.34,A -85,B 0,C 180,E1 -6727.066,E2 -6727.066} C_VEL
LIN {X 0,Y 481.725,Z 464.467,A -85,B 0,C 180,E1 -6727.761,E2 -6727.761} C_VEL
LIN {X 0,Y 481.636,Z 464.478,A -85,B 0,C 180,E1 -6727.997,E2 -6727.997} C_VEL
LIN {X 0,Y 481.71,Z 464.48,A -85,B 0,C 180,E1 -6730.394,E2 -6730.394} C_VEL
LIN {X 0,Y 481.729,Z 464.502,A -85,B 0,C 180,E1 -6733.69,E2 -6733.69} C_VEL
LIN {X 0,Y 481.879,Z 465.219,A -85,B 0,C 180,E1 -6733.899,E2 -6733.899} C_VEL
LIN {X 0,Y 483.629,Z 470.193,A -85,B 0,C 180,E1 -6734.075,E2 -6734.075} C_VEL
LIN {X 0,Y 485.102,Z 474.917,A -85,B 0,C 180,E1 -6734.2,E2 -6734.2} C_VEL
LIN {X 0,Y 484.691,Z 545.451,A -85,B 0,C 180,E1 -6735.274,E2 -6735.274} C_VEL
LIN {X 0,Y 484.633,Z 558.512,A -85,B 0,C 180,E1 -6735.648,E2 -6735.648} C_VEL
LIN {X 0,Y 484.429,Z 570.515,A -85,B 0,C 180,E1 -6736.151,E2 -6736.151} C_VEL
LIN {X 0,Y 484.186,Z 581.769,A -85,B 0,C 180,E1 -6736.783,E2 -6736.783} C_VEL
LIN {X 0,Y 483.73,Z 593.364,A -85,B 0,C 180,E1 -6737.626,E2 -6737.626} C_VEL
LIN {X 0,Y 483.325,Z 603.708,A -85,B 0,C 180,E1 -6738.573,E2 -6738.573} C_VEL
LIN {X 0,Y 482.959,Z 612.147,A -85,B 0,C 180,E1 -6739.52,E2 -6739.52} C_VEL
LIN {X 0,Y 482.677,Z 619.896,A -85,B 0,C 180,E1 -6740.572,E2 -6740.572} C_VEL
LIN {X 0,Y 482.282,Z 627.587,A -85,B 0,C 180,E1 -6741.853,E2 -6741.853} C_VEL
LIN {X 0,Y 482.041,Z 633.346,A -85,B 0,C 180,E1 -6743.049,E2 -6743.049} C_VEL
LIN {X 0,Y 481.906,Z 637.624,A -85,B 0,C 180,E1 -6744.141,E2 -6744.141} C_VEL
LIN {X 0,Y 481.659,Z 641.514,A -85,B 0,C 180,E1 -6745.397,E2 -6745.397} C_VEL
LIN {X 0,Y 481.493,Z 644.383,A -85,B 0,C 180,E1 -6746.653,E2 -6746.653} C_VEL
LIN {X 0,Y 481.514,Z 645.747,A -85,B 0,C 180,E1 -6747.49,E2 -6747.49} C_VEL
LIN {X 0,Y 481.398,Z 646.733,A -85,B 0,C 180,E1 -6748.327,E2 -6748.327} C_VEL
LIN {X 0,Y 481.469,Z 647.322,A -85,B 0,C 180,E1 -6749.164,E2 -6749.164} C_VEL
LIN {X 0,Y 481.454,Z 647.555,A -85,B 0,C 180,E1 -6750,E2 -6750} C_VEL
LIN {X 0,Y 481.469,Z 647.372,A -85,B 0,C 180,E1 -6750.836,E2 -6750.836} C_VEL
LIN {X 0,Y 481.398,Z 646.816,A -85,B 0,C 180,E1 -6751.673,E2 -6751.673} C_VEL
LIN {X 0,Y 481.513,Z 645.862,A -85,B 0,C 180,E1 -6752.51,E2 -6752.51} C_VEL
LIN {X 0,Y 481.488,Z 644.55,A -85,B 0,C 180,E1 -6753.347,E2 -6753.347} C_VEL
LIN {X 0,Y 481.655,Z 641.743,A -85,B 0,C 180,E1 -6754.603,E2 -6754.603} C_VEL
LIN {X 0,Y 481.896,Z 637.931,A -85,B 0,C 180,E1 -6755.859,E2 -6755.859} C_VEL
LIN {X 0,Y 482.007,Z 632.85,A -85,B 0,C 180,E1 -6757.163,E2 -6757.163} C_VEL
LIN {X 0,Y 482.301,Z 626.842,A -85,B 0,C 180,E1 -6758.379,E2 -6758.379} C_VEL
LIN {X 0,Y 482.728,Z 619.069,A -85,B 0,C 180,E1 -6759.638,E2 -6759.638} C_VEL
LIN {X 0,Y 483.096,Z 609.405,A -85,B 0,C 180,E1 -6760.901,E2 -6760.901} C_VEL
LIN {X 0,Y 483.492,Z 600.381,A -85,B 0,C 180,E1 -6761.848,E2 -6761.848} C_VEL
LIN {X 0,Y 483.929,Z 589.898,A -85,B 0,C 180,E1 -6762.737,E2 -6762.737} C_VEL
LIN {X 0,Y 484.227,Z 578.407,A -85,B 0,C 180,E1 -6763.514,E2 -6763.514} C_VEL
LIN {X 0,Y 484.441,Z 567.183,A -85,B 0,C 180,E1 -6764.101,E2 -6764.101} C_VEL
LIN {X 0,Y 484.649,Z 554.029,A -85,B 0,C 180,E1 -6764.593,E2 -6764.593} C_VEL
LIN {X 0,Y 484.676,Z 540.35,A -85,B 0,C 180,E1 -6764.914,E2 -6764.914} C_VEL
LIN {X 0,Y 485.005,Z 473.905,A -85,B 0,C 180,E1 -6765.911,E2 -6765.911} C_VEL
LIN {X 0,Y 481.869,Z 465.306,A -85,B 0,C 180,E1 -6766.185,E2 -6766.185} C_VEL
LIN {X 0,Y 481.701,Z 464.552,A -85,B 0,C 180,E1 -6766.349,E2 -6766.349} C_VEL
LIN {X 0,Y 481.715,Z 464.458,A -85,B 0,C 180,E1 -6768.721,E2 -6768.721} C_VEL
LIN {X 0,Y 481.647,Z 464.481,A -85,B 0,C 180,E1 -6771.394,E2 -6771.394} C_VEL
LIN {X 0,Y 481.675,Z 464.483,A -85,B 0,C 180,E1 -6774.113,E2 -6774.113} C_VEL
LIN {X 0,Y 481.747,Z 464.46,A -85,B 0,C 180,E1 -6777.138,E2 -6777.138} C_VEL
LIN {X 0,Y 481.679,Z 464.482,A -85,B 0,C 180,E1 -6779.74,E2 -6779.74} C_VEL
LIN {X 0,Y 481.672,Z 464.481,A -85,B 0,C 180,E1 -6782.673,E2 -6782.673} C_VEL
LIN {X 0,Y 481.639,Z 464.484,A -85,B 0,C 180,E1 -6785.708,E2 -6785.708} C_VEL
LIN {X 0,Y 481.669,Z 464.486,A -85,B 0,C 180,E1 -6788.858,E2 -6788.858} C_VEL
LIN {X 0,Y 481.659,Z 464.476,A -85,B 0,C 180,E1 -6791.913,E2 -6791.913} C_VEL
LIN {X 0,Y 481.656,Z 464.481,A -85,B 0,C 180,E1 -6794.456,E2 -6794.456} C_VEL
LIN {X 0,Y 481.643,Z 464.482,A -85,B 0,C 180,E1 -6797.839,E2 -6797.839} C_VEL
LIN {X 0,Y 481.656,Z 464.469,A -85,B 0,C 180,E1 -6800.653,E2 -6800.653} C_VEL
LIN {X 0,Y 481.626,Z 464.493,A -85,B 0,C 180,E1 -6803.375,E2 -6803.375} C_VEL
LIN {X 0,Y 481.703,Z 464.475,A -85,B 0,C 180,E1 -6806.329,E2 -6806.329} C_VEL
LIN {X 0,Y 481.651,Z 464.469,A -85,B 0,C 180,E1 -6809.415,E2 -6809.415} C_VEL
LIN {X 0,Y 481.695,Z 464.474,A -85,B 0,C 180,E1 -6812.168,E2 -6812.168} C_VEL
LIN {X 0,Y 481.71,Z 464.481,A -85,B 0,C 180,E1 -6814.969,E2 -6814.969} C_VEL
LIN {X 0,Y 481.642,Z 464.484,A -85,B 0,C 180,E1 -6817.704,E2 -6817.704} C_VEL
LIN {X 0,Y 481.699,Z 464.478,A -85,B 0,C 180,E1 -6820.393,E2 -6820.393} C_VEL
LIN {X 0,Y 481.683,Z 464.483,A -85,B 0,C 180,E1 -6823.034,E2 -6823.034} C_VEL
LIN {X 0,Y 481.685,Z 464.484,A -85,B 0,C 180,E1 -6825.638,E2 -6825.638} C_VEL
LIN {X 0,Y 481.743,Z 464.471,A -85,B 0,C 180,E1 -6828.215,E2 -6828.215} C_VEL
LIN {X 0,Y 481.754,Z 464.474,A -85,B 0,C 180,E1 -6831.611,E2 -6831.611} C_VEL
LIN {X 0,Y 481.808,Z 464.464,A -85,B 0,C 180,E1 -6834.139,E2 -6834.139} C_VEL
LIN {X 0,Y 481.919,Z 464.449,A -85,B 0,C 180,E1 -6837.492,E2 -6837.492} C_VEL
LIN {X 0,Y 481.93,Z 464.449,A -85,B 0,C 180,E1 -6840,E2 -6840} C_VEL
LIN {X 0,Y 481.919,Z 464.447,A -85,B 0,C 180,E1 -6842.507,E2 -6842.507} C_VEL
LIN {X 0,Y 481.819,Z 464.465,A -85,B 0,C 180,E1 -6845.86,E2 -6845.86} C_VEL
LIN {X 0,Y 481.754,Z 464.47,A -85,B 0,C 180,E1 -6848.388,E2 -6848.388} C_VEL
LIN {X 0,Y 481.743,Z 464.475,A -85,B 0,C 180,E1 -6851.785,E2 -6851.785} C_VEL
LIN {X 0,Y 481.733,Z 464.478,A -85,B 0,C 180,E1 -6855.225,E2 -6855.225} C_VEL
LIN {X 0,Y 481.703,Z 464.464,A -85,B 0,C 180,E1 -6858.722,E2 -6858.722} C_VEL
LIN {X 0,Y 481.637,Z 464.486,A -85,B 0,C 180,E1 -6861.395,E2 -6861.395} C_VEL
LIN {X 0,Y 481.668,Z 464.483,A -85,B 0,C 180,E1 -6864.114,E2 -6864.114} C_VEL
LIN {X 0,Y 481.744,Z 464.464,A -85,B 0,C 180,E1 -6867.141,E2 -6867.141} C_VEL
LIN {X 0,Y 481.681,Z 464.488,A -85,B 0,C 180,E1 -6869.741,E2 -6869.741} C_VEL
LIN {X 0,Y 481.666,Z 464.476,A -85,B 0,C 180,E1 -6872.675,E2 -6872.675} C_VEL
LIN {X 0,Y 481.637,Z 464.494,A -85,B 0,C 180,E1 -6875.71,E2 -6875.71} C_VEL
LIN {X 0,Y 481.665,Z 464.48,A -85,B 0,C 180,E1 -6878.86,E2 -6878.86} C_VEL
LIN {X 0,Y 481.648,Z 464.484,A -85,B 0,C 180,E1 -6881.914,E2 -6881.914} C_VEL
LIN {X 0,Y 481.655,Z 464.476,A -85,B 0,C 180,E1 -6884.458,E2 -6884.458} C_VEL
LIN {X 0,Y 481.684,Z 464.481,A -85,B 0,C 180,E1 -6886.847,E2 -6886.847} C_VEL
LIN {X 0,Y 481.686,Z 464.478,A -85,B 0,C 180,E1 -6890.062,E2 -6890.062} C_VEL
LIN {X 0,Y 481.626,Z 464.487,A -85,B 0,C 180,E1 -6893.254,E2 -6893.254} C_VEL
LIN {X 0,Y 481.708,Z 464.476,A -85,B 0,C 180,E1 -6896.331,E2 -6896.331} C_VEL
LIN {X 0,Y 481.739,Z 464.584,A -85,B 0,C 180,E1 -6900.113,E2 -6900.113} C_VEL
LIN {X 0,Y 483.917,Z 474.324,A -85,B 0,C 180,E1 -6901.59,E2 -6901.59} C_VEL
LIN {X 0,Y 485.234,Z 481.598,A -85,B 0,C 180,E1 -6902.623,E2 -6902.623} C_VEL
LIN {X 0,Y 484.337,Z 506.125,A -85,B 0,C 180,E1 -6905.801,E2 -6905.801} C_VEL
LIN {X 0,Y 483.485,Z 530.546,A -85,B 0,C 180,E1 -6908.915,E2 -6908.915} C_VEL
LIN {X 0,Y 482.738,Z 554.677,A -85,B 0,C 180,E1 -6911.979,E2 -6911.979} C_VEL
LIN {X 0,Y 482.447,Z 566.469,A -85,B 0,C 180,E1 -6913.454,E2 -6913.454} C_VEL
LIN {X 0,Y 484.704,Z 588.557,A -85,B 0,C 180,E1 -6913.877,E2 -6913.877} C_VEL
LIN {X 0,Y 484.115,Z 676.822,A -85,B 0,C 180,E1 -6915.202,E2 -6915.202} C_VEL
LIN {X 0,Y 483.795,Z 690.175,A -85,B 0,C 180,E1 -6915.569,E2 -6915.569} C_VEL
LIN {X 0,Y 483.366,Z 702.431,A -85,B 0,C 180,E1 -6916.066,E2 -6916.066} C_VEL
LIN {X 0,Y 482.915,Z 714.841,A -85,B 0,C 180,E1 -6916.75,E2 -6916.75} C_VEL
LIN {X 0,Y 482.473,Z 726.298,A -85,B 0,C 180,E1 -6917.569,E2 -6917.569} C_VEL
LIN {X 0,Y 481.978,Z 737.184,A -85,B 0,C 180,E1 -6918.541,E2 -6918.541} C_VEL
LIN {X 0,Y 481.711,Z 745.886,A -85,B 0,C 180,E1 -6919.492,E2 -6919.492} C_VEL
LIN {X 0,Y 481.45,Z 753.93,A -85,B 0,C 180,E1 -6920.548,E2 -6920.548} C_VEL
LIN {X 0,Y 481.252,Z 761.81,A -85,B 0,C 180,E1 -6921.814,E2 -6921.814} C_VEL
LIN {X 0,Y 481.082,Z 769.081,A -85,B 0,C 180,E1 -6923.289,E2 -6923.289} C_VEL
LIN {X 0,Y 481.074,Z 773.94,A -85,B 0,C 180,E1 -6924.551,E2 -6924.551} C_VEL
LIN {X 0,Y 481.077,Z 777.658,A -85,B 0,C 180,E1 -6925.811,E2 -6925.811} C_VEL
LIN {X 0,Y 481.058,Z 779.573,A -85,B 0,C 180,E1 -6926.65,E2 -6926.65} C_VEL
LIN {X 0,Y 481.048,Z 781.011,A -85,B 0,C 180,E1 -6927.488,E2 -6927.488} C_VEL
LIN {X 0,Y 481.089,Z 782.67,A -85,B 0,C 180,E1 -6929.163,E2 -6929.163} C_VEL
LIN {X 0,Y 481.093,Z 782.893,A -85,B 0,C 180,E1 -6930,E2 -6930} C_VEL
LIN {X 0,Y 481.089,Z 782.671,A -85,B 0,C 180,E1 -6930.837,E2 -6930.837} C_VEL
LIN {X 0,Y 481.048,Z 781.015,A -85,B 0,C 180,E1 -6932.512,E2 -6932.512} C_VEL
LIN {X 0,Y 481.058,Z 779.577,A -85,B 0,C 180,E1 -6933.35,E2 -6933.35} C_VEL
LIN {X 0,Y 481.043,Z 776.553,A -85,B 0,C 180,E1 -6934.609,E2 -6934.609} C_VEL
LIN {X 0,Y 481.125,Z 772.474,A -85,B 0,C 180,E1 -6935.869,E2 -6935.869} C_VEL
LIN {X 0,Y 481.153,Z 766.191,A -85,B 0,C 180,E1 -6937.343,E2 -6937.343} C_VEL
LIN {X 0,Y 481.305,Z 759.354,A -85,B 0,C 180,E1 -6938.608,E2 -6938.608} C_VEL
LIN {X 0,Y 481.52,Z 750.887,A -85,B 0,C 180,E1 -6939.875,E2 -6939.875} C_VEL
LIN {X 0,Y 481.849,Z 742.236,A -85,B 0,C 180,E1 -6940.93,E2 -6940.93} C_VEL
LIN {X 0,Y 482.235,Z 732.905,A -85,B 0,C 180,E1 -6941.867,E2 -6941.867} C_VEL
LIN {X 0,Y 482.666,Z 721.057,A -85,B 0,C 180,E1 -6942.829,E2 -6942.829} C_VEL
LIN {X 0,Y 483.061,Z 709.548,A -85,B 0,C 180,E1 -6943.568,E2 -6943.568} C_VEL
LIN {X 0,Y 483.51,Z 697.778,A -85,B 0,C 180,E1 -6944.145,E2 -6944.145} C_VEL
LIN {X 0,Y 483.932,Z 685.182,A -85,B 0,C 180,E1 -6944.588,E2 -6944.588} C_VEL
LIN {X 0,Y 484.194,Z 672.458,A -85,B 0,C 180,E1 -6944.876,E2 -6944.876} C_VEL
LIN {X 0,Y 484.646,Z 586.192,A -85,B 0,C 180,E1 -6946.16,E2 -6946.16} C_VEL
LIN {X 0,Y 482.443,Z 566.465,A -85,B 0,C 180,E1 -6946.546,E2 -6946.546} C_VEL
LIN {X 0,Y 483.135,Z 540.916,A -85,B 0,C 180,E1 -6949.767,E2 -6949.767} C_VEL
LIN {X 0,Y 483.887,Z 518.354,A -85,B 0,C 180,E1 -6952.636,E2 -6952.636} C_VEL
LIN {X 0,Y 484.669,Z 495.599,A -85,B 0,C 180,E1 -6955.555,E2 -6955.555} C_VEL
LIN {X 0,Y 485.202,Z 481.582,A -85,B 0,C 180,E1 -6957.379,E2 -6957.379} C_VEL
LIN {X 0,Y 484.295,Z 476.052,A -85,B 0,C 180,E1 -6958.158,E2 -6958.158} C_VEL
LIN {X 0,Y 481.723,Z 464.609,A -85,B 0,C 180,E1 -6959.873,E2 -6959.873} C_VEL
LIN {X 0,Y 481.67,Z 464.483,A -85,B 0,C 180,E1 -6962.673,E2 -6962.673} C_VEL
LIN {X 0,Y 481.634,Z 464.489,A -85,B 0,C 180,E1 -6965.709,E2 -6965.709} C_VEL
LIN {X 0,Y 481.711,Z 464.476,A -85,B 0,C 180,E1 -6969.353,E2 -6969.353} C_VEL
LIN {X 0,Y 481.67,Z 464.486,A -85,B 0,C 180,E1 -6972.157,E2 -6972.157} C_VEL
LIN {X 0,Y 481.656,Z 464.48,A -85,B 0,C 180,E1 -6974.456,E2 -6974.456} C_VEL
LIN {X 0,Y 481.643,Z 464.481,A -85,B 0,C 180,E1 -6977.839,E2 -6977.839} C_VEL
LIN {X 0,Y 481.675,Z 464.481,A -85,B 0,C 180,E1 -6980.65,E2 -6980.65} C_VEL
LIN {X 0,Y 481.625,Z 464.487,A -85,B 0,C 180,E1 -6983.375,E2 -6983.375} C_VEL
LIN {X 0,Y 481.703,Z 464.478,A -85,B 0,C 180,E1 -6986.329,E2 -6986.329} C_VEL
LIN {X 0,Y 481.651,Z 464.484,A -85,B 0,C 180,E1 -6989.415,E2 -6989.415} C_VEL
LIN {X 0,Y 481.695,Z 464.479,A -85,B 0,C 180,E1 -6992.168,E2 -6992.168} C_VEL
LIN {X 0,Y 481.71,Z 464.477,A -85,B 0,C 180,E1 -6994.969,E2 -6994.969} C_VEL
LIN {X 0,Y 481.641,Z 464.486,A -85,B 0,C 180,E1 -6997.704,E2 -6997.704} C_VEL
LIN {X 0,Y 481.699,Z 464.472,A -85,B 0,C 180,E1 -7000.393,E2 -7000.393} C_VEL
LIN {X 0,Y 481.683,Z 464.478,A -85,B 0,C 180,E1 -7003.034,E2 -7003.034} C_VEL
LIN {X 0,Y 481.68,Z 464.481,A -85,B 0,C 180,E1 -7005.638,E2 -7005.638} C_VEL
LIN {X 0,Y 481.743,Z 464.475,A -85,B 0,C 180,E1 -7008.215,E2 -7008.215} C_VEL
LIN {X 0,Y 481.754,Z 464.471,A -85,B 0,C 180,E1 -7011.612,E2 -7011.612} C_VEL
LIN {X 0,Y 481.819,Z 464.465,A -85,B 0,C 180,E1 -7014.14,E2 -7014.14} C_VEL
LIN {X 0,Y 481.92,Z 464.449,A -85,B 0,C 180,E1 -7017.493,E2 -7017.493} C_VEL
LIN {X 0,Y 481.93,Z 464.45,A -85,B 0,C 180,E1 -7020,E2 -7020} C_VEL
LIN {X 0,Y 481.919,Z 464.45,A -85,B 0,C 180,E1 -7022.508,E2 -7022.508} C_VEL
LIN {X 0,Y 481.822,Z 464.462,A -85,B 0,C 180,E1 -7025.86,E2 -7025.86} C_VEL
LIN {X 0,Y 481.754,Z 464.474,A -85,B 0,C 180,E1 -7028.389,E2 -7028.389} C_VEL
LIN {X 0,Y 481.743,Z 464.471,A -85,B 0,C 180,E1 -7031.785,E2 -7031.785} C_VEL
LIN {X 0,Y 481.735,Z 464.47,A -85,B 0,C 180,E1 -7035.225,E2 -7035.225} C_VEL
LIN {X 0,Y 481.704,Z 464.484,A -85,B 0,C 180,E1 -7038.722,E2 -7038.722} C_VEL
LIN {X 0,Y 481.639,Z 464.482,A -85,B 0,C 180,E1 -7041.395,E2 -7041.395} C_VEL
LIN {X 0,Y 481.669,Z 464.481,A -85,B 0,C 180,E1 -7044.114,E2 -7044.114} C_VEL
LIN {X 0,Y 481.744,Z 464.472,A -85,B 0,C 180,E1 -7047.141,E2 -7047.141} C_VEL
LIN {X 0,Y 481.681,Z 464.464,A -85,B 0,C 180,E1 -7049.741,E2 -7049.741} C_VEL
LIN {X 0,Y 481.667,Z 464.474,A -85,B 0,C 180,E1 -7052.675,E2 -7052.675} C_VEL
LIN {X 0,Y 481.637,Z 464.486,A -85,B 0,C 180,E1 -7055.71,E2 -7055.71} C_VEL
LIN {X 0,Y 481.666,Z 464.476,A -85,B 0,C 180,E1 -7058.86,E2 -7058.86} C_VEL
LIN {X 0,Y 481.648,Z 464.48,A -85,B 0,C 180,E1 -7061.914,E2 -7061.914} C_VEL
LIN {X 0,Y 481.655,Z 464.486,A -85,B 0,C 180,E1 -7064.458,E2 -7064.458} C_VEL
LIN {X 0,Y 481.651,Z 464.477,A -85,B 0,C 180,E1 -7067.841,E2 -7067.841} C_VEL
LIN {X 0,Y 481.69,Z 464.484,A -85,B 0,C 180,E1 -7071.144,E2 -7071.144} C_VEL
LIN {X 0,Y 481.665,Z 464.461,A -85,B 0,C 180,E1 -7074.796,E2 -7074.796} C_VEL
LIN {X 0,Y 481.672,Z 464.474,A -85,B 0,C 180,E1 -7077.327,E2 -7077.327} C_VEL
LIN {X 0,Y 481.679,Z 464.483,A -85,B 0,C 180,E1 -7080.26,E2 -7080.26} C_VEL
LIN {X 0,Y 481.746,Z 464.461,A -85,B 0,C 180,E1 -7083.113,E2 -7083.113} C_VEL
LIN {X 0,Y 481.675,Z 464.483,A -85,B 0,C 180,E1 -7085.887,E2 -7085.887} C_VEL
LIN {X 0,Y 481.636,Z 464.478,A -85,B 0,C 180,E1 -7087.997,E2 -7087.997} C_VEL
LIN {X 0,Y 480.97,Z 464.566,A -85,B 0,C 180,E1 -7088.695,E2 -7088.695} C_VEL
LIN {X 0,Y 478.144,Z 464.925,A -85,B 0,C 180,E1 -7089.829,E2 -7089.829} C_VEL
LIN {X 0,Y 475.759,Z 465.212,A -85,B 0,C 180,E1 -7090.743,E2 -7090.743} C_VEL
LIN {X 0,Y 474.738,Z 465.325,A -85,B 0,C 180,E1 -7091.449,E2 -7091.449} C_VEL
LIN {X 0,Y 474.656,Z 465.329,A -85,B 0,C 180,E1 -7091.688,E2 -7091.688} C_VEL
LIN {X 0,Y 474.697,Z 465.48,A -85,B 0,C 180,E1 -7093.524,E2 -7093.524} C_VEL
LIN {X 0,Y 474.944,Z 466.512,A -85,B 0,C 180,E1 -7093.684,E2 -7093.684} C_VEL
LIN {X 0,Y 478.307,Z 476.151,A -85,B 0,C 180,E1 -7093.973,E2 -7093.973} C_VEL
LIN {X 0,Y 477.882,Z 546.46,A -85,B 0,C 180,E1 -7095.059,E2 -7095.059} C_VEL
LIN {X 0,Y 477.816,Z 559.515,A -85,B 0,C 180,E1 -7095.439,E2 -7095.439} C_VEL
LIN {X 0,Y 477.601,Z 571.514,A -85,B 0,C 180,E1 -7095.949,E2 -7095.949} C_VEL
LIN {X 0,Y 477.341,Z 583.166,A -85,B 0,C 180,E1 -7096.617,E2 -7096.617} C_VEL
LIN {X 0,Y 476.866,Z 594.358,A -85,B 0,C 180,E1 -7097.445,E2 -7097.445} C_VEL
LIN {X 0,Y 476.438,Z 604.701,A -85,B 0,C 180,E1 -7098.406,E2 -7098.406} C_VEL
LIN {X 0,Y 476.052,Z 613.139,A -85,B 0,C 180,E1 -7099.366,E2 -7099.366} C_VEL
LIN {X 0,Y 475.746,Z 620.887,A -85,B 0,C 180,E1 -7100.434,E2 -7100.434} C_VEL
LIN {X 0,Y 475.327,Z 628.578,A -85,B 0,C 180,E1 -7101.733,E2 -7101.733} C_VEL
LIN {X 0,Y 475.065,Z 634.336,A -85,B 0,C 180,E1 -7102.946,E2 -7102.946} C_VEL
LIN {X 0,Y 474.921,Z 638.613,A -85,B 0,C 180,E1 -7104.054,E2 -7104.054} C_VEL
LIN {X 0,Y 474.651,Z 642.504,A -85,B 0,C 180,E1 -7105.329,E2 -7105.329} C_VEL
LIN {X 0,Y 474.474,Z 645.373,A -85,B 0,C 180,E1 -7106.603,E2 -7106.603} C_VEL
LIN {X 0,Y 474.499,Z 646.735,A -85,B 0,C 180,E1 -7107.453,E2 -7107.453} C_VEL
LIN {X 0,Y 474.377,Z 647.721,A -85,B 0,C 180,E1 -7108.302,E2 -7108.302} C_VEL
LIN {X 0,Y 474.451,Z 648.309,A -85,B 0,C 180,E1 -7109.151,E2 -7109.151} C_VEL
LIN {X 0,Y 474.435,Z 648.541,A -85,B 0,C 180,E1 -7110,E2 -7110} C_VEL
LIN {X 0,Y 474.451,Z 648.359,A -85,B 0,C 180,E1 -7110.849,E2 -7110.849} C_VEL
LIN {X 0,Y 474.377,Z 647.803,A -85,B 0,C 180,E1 -7111.698,E2 -7111.698} C_VEL
LIN {X 0,Y 474.498,Z 646.849,A -85,B 0,C 180,E1 -7112.547,E2 -7112.547} C_VEL
LIN {X 0,Y 474.469,Z 645.538,A -85,B 0,C 180,E1 -7113.397,E2 -7113.397} C_VEL
LIN {X 0,Y 474.646,Z 642.731,A -85,B 0,C 180,E1 -7114.671,E2 -7114.671} C_VEL
LIN {X 0,Y 474.911,Z 638.917,A -85,B 0,C 180,E1 -7115.946,E2 -7115.946} C_VEL
LIN {X 0,Y 475.034,Z 633.839,A -85,B 0,C 180,E1 -7117.268,E2 -7117.268} C_VEL
LIN {X 0,Y 475.352,Z 627.828,A -85,B 0,C 180,E1 -7118.502,E2 -7118.502} C_VEL
LIN {X 0,Y 475.803,Z 620.054,A -85,B 0,C 180,E1 -7119.78,E2 -7119.78} C_VEL
LIN {X 0,Y 476.195,Z 610.39,A -85,B 0,C 180,E1 -7121.061,E2 -7121.061} C_VEL
LIN {X 0,Y 476.615,Z 601.365,A -85,B 0,C 180,E1 -7122.021,E2 -7122.021} C_VEL
LIN {X 0,Y 477.077,Z 590.88,A -85,B 0,C 180,E1 -7122.923,E2 -7122.923} C_VEL
LIN {X 0,Y 477.396,Z 579.388,A -85,B 0,C 180,E1 -7123.711,E2 -7123.711} C_VEL
LIN {X 0,Y 477.641,Z 568.16,A -85,B 0,C 180,E1 -7124.306,E2 -7124.306} C_VEL
LIN {X 0,Y 477.834,Z 555.005,A -85,B 0,C 180,E1 -7124.806,E2 -7124.806} C_VEL
LIN {X 0,Y 477.862,Z 541.317,A -85,B 0,C 180,E1 -7125.132,E2 -7125.132} C_VEL
LIN {X 0,Y 478.245,Z 475.504,A -85,B 0,C 180,E1 -7126.132,E2 -7126.132} C_VEL
LIN {X 0,Y 474.831,Z 466.206,A -85,B 0,C 180,E1 -7126.432,E2 -7126.432} C_VEL
LIN {X 0,Y 474.659,Z 465.432,A -85,B 0,C 180,E1 -7126.598,E2 -7126.598} C_VEL
LIN {X 0,Y 474.668,Z 465.34,A -85,B 0,C 180,E1 -7129.01,E2 -7129.01} C_VEL
LIN {X 0,Y 474.59,Z 465.357,A -85,B 0,C 180,E1 -7131.728,E2 -7131.728} C_VEL
LIN {X 0,Y 474.658,Z 465.359,A -85,B 0,C 180,E1 -7134.492,E2 -7134.492} C_VEL
LIN {X 0,Y 474.681,Z 465.339,A -85,B 0,C 180,E1 -7137.334,E2 -7137.334} C_VEL
LIN {X 0,Y 474.605,Z 465.369,A -85,B 0,C 180,E1 -7140.81,E2 -7140.81} C_VEL
LIN {X 0,Y 474.637,Z 465.358,A -85,B 0,C 180,E1 -7143.983,E2 -7143.983} C_VEL
LIN {X 0,Y 474.572,Z 465.365,A -85,B 0,C 180,E1 -7146.899,E2 -7146.899} C_VEL
LIN {X 0,Y 474.625,Z 465.362,A -85,B 0,C 180,E1 -7149.647,E2 -7149.647} C_VEL
LIN {X 0,Y 474.632,Z 465.353,A -85,B 0,C 180,E1 -7152.931,E2 -7152.931} C_VEL
LIN {X 0,Y 474.605,Z 465.363,A -85,B 0,C 180,E1 -7155.894,E2 -7155.894} C_VEL
LIN {X 0,Y 474.623,Z 465.353,A -85,B 0,C 180,E1 -7159.04,E2 -7159.04} C_VEL
LIN {X 0,Y 474.605,Z 465.359,A -85,B 0,C 180,E1 -7161.703,E2 -7161.703} C_VEL
LIN {X 0,Y 474.624,Z 465.362,A -85,B 0,C 180,E1 -7164.725,E2 -7164.725} C_VEL
LIN {X 0,Y 474.631,Z 465.346,A -85,B 0,C 180,E1 -7167.787,E2 -7167.787} C_VEL
LIN {X 0,Y 474.625,Z 465.346,A -85,B 0,C 180,E1 -7170.882,E2 -7170.882} C_VEL
LIN {X 0,Y 474.659,Z 465.358,A -85,B 0,C 180,E1 -7173.628,E2 -7173.628} C_VEL
LIN {X 0,Y 474.627,Z 465.358,A -85,B 0,C 180,E1 -7176.641,E2 -7176.641} C_VEL
LIN {X 0,Y 474.648,Z 465.357,A -85,B 0,C 180,E1 -7180.089,E2 -7180.089} C_VEL
LIN {X 0,Y 474.642,Z 465.357,A -85,B 0,C 180,E1 -7182.774,E2 -7182.774} C_VEL
LIN {X 0,Y 474.643,Z 465.362,A -85,B 0,C 180,E1 -7185.421,E2 -7185.421} C_VEL
LIN {X 0,Y 474.696,Z 465.35,A -85,B 0,C 180,E1 -7188.037,E2 -7188.037} C_VEL
LIN {X 0,Y 474.72,Z 465.349,A -85,B 0,C 180,E1 -7191.486,E2 -7191.486} C_VEL
LIN {X 0,Y 474.77,Z 465.341,A -85,B 0,C 180,E1 -7194.052,E2 -7194.052} C_VEL
LIN {X 0,Y 474.886,Z 465.325,A -85,B 0,C 180,E1 -7197.455,E2 -7197.455} C_VEL
LIN {X 0,Y 474.867,Z 465.329,A -85,B 0,C 180,E1 -7200.848,E2 -7200.848} C_VEL
LIN {X 0,Y 474.886,Z 465.323,A -85,B 0,C 180,E1 -7202.545,E2 -7202.545} C_VEL
LIN {X 0,Y 474.78,Z 465.341,A -85,B 0,C 180,E1 -7205.948,E2 -7205.948} C_VEL
LIN {X 0,Y 474.719,Z 465.346,A -85,B 0,C 180,E1 -7208.514,E2 -7208.514} C_VEL
LIN {X 0,Y 474.696,Z 465.351,A -85,B 0,C 180,E1 -7211.963,E2 -7211.963} C_VEL
LIN {X 0,Y 474.69,Z 465.358,A -85,B 0,C 180,E1 -7215.456,E2 -7215.456} C_VEL
LIN {X 0,Y 474.657,Z 465.343,A -85,B 0,C 180,E1 -7219.011,E2 -7219.011} C_VEL
LIN {X 0,Y 474.581,Z 465.371,A -85,B 0,C 180,E1 -7221.729,E2 -7221.729} C_VEL
LIN {X 0,Y 474.651,Z 465.355,A -85,B 0,C 180,E1 -7224.493,E2 -7224.493} C_VEL
LIN {X 0,Y 474.691,Z 465.344,A -85,B 0,C 180,E1 -7227.339,E2 -7227.339} C_VEL
LIN {X 0,Y 474.603,Z 465.362,A -85,B 0,C 180,E1 -7230.812,E2 -7230.812} C_VEL
LIN {X 0,Y 474.632,Z 465.362,A -85,B 0,C 180,E1 -7233.985,E2 -7233.985} C_VEL
LIN {X 0,Y 474.569,Z 465.366,A -85,B 0,C 180,E1 -7236.901,E2 -7236.901} C_VEL
LIN {X 0,Y 474.622,Z 465.364,A -85,B 0,C 180,E1 -7239.648,E2 -7239.648} C_VEL
LIN {X 0,Y 474.61,Z 465.354,A -85,B 0,C 180,E1 -7242.935,E2 -7242.935} C_VEL
LIN {X 0,Y 474.614,Z 465.363,A -85,B 0,C 180,E1 -7245.897,E2 -7245.897} C_VEL
LIN {X 0,Y 474.643,Z 465.353,A -85,B 0,C 180,E1 -7249.039,E2 -7249.039} C_VEL
LIN {X 0,Y 474.614,Z 465.368,A -85,B 0,C 180,E1 -7251.704,E2 -7251.704} C_VEL
LIN {X 0,Y 474.626,Z 465.362,A -85,B 0,C 180,E1 -7254.727,E2 -7254.727} C_VEL
LIN {X 0,Y 474.636,Z 465.365,A -85,B 0,C 180,E1 -7257.789,E2 -7257.789} C_VEL
LIN {X 0,Y 474.694,Z 465.568,A -85,B 0,C 180,E1 -7259.911,E2 -7259.911} C_VEL
LIN {X 0,Y 478.177,Z 481.419,A -85,B 0,C 180,E1 -7262.283,E2 -7262.283} C_VEL
LIN {X 0,Y 478.185,Z 487.912,A -85,B 0,C 180,E1 -7263.156,E2 -7263.156} C_VEL
LIN {X 0,Y 477.171,Z 512.607,A -85,B 0,C 180,E1 -7266.392,E2 -7266.392} C_VEL
LIN {X 0,Y 476.35,Z 534.806,A -85,B 0,C 180,E1 -7269.263,E2 -7269.263} C_VEL
LIN {X 0,Y 475.615,Z 558.817,A -85,B 0,C 180,E1 -7272.367,E2 -7272.367} C_VEL
LIN {X 0,Y 475.45,Z 565.473,A -85,B 0,C 180,E1 -7273.203,E2 -7273.203} C_VEL
LIN {X 0,Y 477.87,Z 588.429,A -85,B 0,C 180,E1 -7273.653,E2 -7273.653} C_VEL
LIN {X 0,Y 477.256,Z 675.829,A -85,B 0,C 180,E1 -7274.985,E2 -7274.985} C_VEL
LIN {X 0,Y 476.891,Z 689.175,A -85,B 0,C 180,E1 -7275.355,E2 -7275.355} C_VEL
LIN {X 0,Y 476.486,Z 700.291,A -85,B 0,C 180,E1 -7275.806,E2 -7275.806} C_VEL
LIN {X 0,Y 475.985,Z 712.116,A -85,B 0,C 180,E1 -7276.444,E2 -7276.444} C_VEL
LIN {X 0,Y 475.529,Z 722.927,A -85,B 0,C 180,E1 -7277.192,E2 -7277.192} C_VEL
LIN {X 0,Y 475.112,Z 734.009,A -85,B 0,C 180,E1 -7278.157,E2 -7278.157} C_VEL
LIN {X 0,Y 474.725,Z 743.059,A -85,B 0,C 180,E1 -7279.12,E2 -7279.12} C_VEL
LIN {X 0,Y 474.401,Z 752.925,A -85,B 0,C 180,E1 -7280.406,E2 -7280.406} C_VEL
LIN {X 0,Y 474.179,Z 760.805,A -85,B 0,C 180,E1 -7281.691,E2 -7281.691} C_VEL
LIN {X 0,Y 474.019,Z 768.081,A -85,B 0,C 180,E1 -7283.188,E2 -7283.188} C_VEL
LIN {X 0,Y 474.016,Z 772.943,A -85,B 0,C 180,E1 -7284.47,E2 -7284.47} C_VEL
LIN {X 0,Y 474.016,Z 776.662,A -85,B 0,C 180,E1 -7285.749,E2 -7285.749} C_VEL
LIN {X 0,Y 474.012,Z 778.581,A -85,B 0,C 180,E1 -7286.6,E2 -7286.6} C_VEL
LIN {X 0,Y 474.005,Z 780.02,A -85,B 0,C 180,E1 -7287.451,E2 -7287.451} C_VEL
LIN {X 0,Y 474.075,Z 781.684,A -85,B 0,C 180,E1 -7289.151,E2 -7289.151} C_VEL
LIN {X 0,Y 474.077,Z 781.907,A -85,B 0,C 180,E1 -7290,E2 -7290} C_VEL
LIN {X 0,Y 474.075,Z 781.685,A -85,B 0,C 180,E1 -7290.849,E2 -7290.849} C_VEL
LIN {X 0,Y 474.005,Z 780.023,A -85,B 0,C 180,E1 -7292.549,E2 -7292.549} C_VEL
LIN {X 0,Y 474.012,Z 778.585,A -85,B 0,C 180,E1 -7293.4,E2 -7293.4} C_VEL
LIN {X 0,Y 473.997,Z 775.559,A -85,B 0,C 180,E1 -7294.677,E2 -7294.677} C_VEL
LIN {X 0,Y 474.06,Z 771.476,A -85,B 0,C 180,E1 -7295.956,E2 -7295.956} C_VEL
LIN {X 0,Y 474.095,Z 765.191,A -85,B 0,C 180,E1 -7297.453,E2 -7297.453} C_VEL
LIN {X 0,Y 474.211,Z 758.345,A -85,B 0,C 180,E1 -7298.737,E2 -7298.737} C_VEL
LIN {X 0,Y 474.474,Z 749.881,A -85,B 0,C 180,E1 -7300.023,E2 -7300.023} C_VEL
LIN {X 0,Y 474.83,Z 741.231,A -85,B 0,C 180,E1 -7301.093,E2 -7301.093} C_VEL
LIN {X 0,Y 475.285,Z 731.108,A -85,B 0,C 180,E1 -7302.116,E2 -7302.116} C_VEL
LIN {X 0,Y 475.668,Z 720.047,A -85,B 0,C 180,E1 -7303.021,E2 -7303.021} C_VEL
LIN {X 0,Y 476.116,Z 708.542,A -85,B 0,C 180,E1 -7303.77,E2 -7303.77} C_VEL
LIN {X 0,Y 476.638,Z 696.779,A -85,B 0,C 180,E1 -7304.353,E2 -7304.353} C_VEL
LIN {X 0,Y 477.042,Z 684.177,A -85,B 0,C 180,E1 -7304.804,E2 -7304.804} C_VEL
LIN {X 0,Y 477.329,Z 671.452,A -85,B 0,C 180,E1 -7305.095,E2 -7305.095} C_VEL
LIN {X 0,Y 477.745,Z 586.534,A -85,B 0,C 180,E1 -7306.379,E2 -7306.379} C_VEL
LIN {X 0,Y 475.446,Z 565.308,A -85,B 0,C 180,E1 -7306.808,E2 -7306.808} C_VEL
LIN {X 0,Y 476.191,Z 539.963,A -85,B 0,C 180,E1 -7310.068,E2 -7310.068} C_VEL
LIN {X 0,Y 476.921,Z 519.171,A -85,B 0,C 180,E1 -7312.757,E2 -7312.757} C_VEL
LIN {X 0,Y 477.751,Z 496.451,A -85,B 0,C 180,E1 -7315.719,E2 -7315.719} C_VEL
LIN {X 0,Y 478.292,Z 482.446,A -85,B 0,C 180,E1 -7317.571,E2 -7317.571} C_VEL
LIN {X 0,Y 475.535,Z 469.047,A -85,B 0,C 180,E1 -7319.54,E2 -7319.54} C_VEL
LIN {X 0,Y 474.661,Z 465.456,A -85,B 0,C 180,E1 -7320.137,E2 -7320.137} C_VEL
LIN {X 0,Y 474.641,Z 465.355,A -85,B 0,C 180,E1 -7323.219,E2 -7323.219} C_VEL
LIN {X 0,Y 474.586,Z 465.363,A -85,B 0,C 180,E1 -7326.323,E2 -7326.323} C_VEL
LIN {X 0,Y 474.648,Z 465.356,A -85,B 0,C 180,E1 -7329.65,E2 -7329.65} C_VEL
LIN {X 0,Y 474.648,Z 465.359,A -85,B 0,C 180,E1 -7332.929,E2 -7332.929} C_VEL
LIN {X 0,Y 474.605,Z 465.351,A -85,B 0,C 180,E1 -7335.894,E2 -7335.894} C_VEL
LIN {X 0,Y 474.623,Z 465.361,A -85,B 0,C 180,E1 -7339.04,E2 -7339.04} C_VEL
LIN {X 0,Y 474.605,Z 465.36,A -85,B 0,C 180,E1 -7341.703,E2 -7341.703} C_VEL
LIN {X 0,Y 474.624,Z 465.361,A -85,B 0,C 180,E1 -7344.726,E2 -7344.726} C_VEL
LIN {X 0,Y 474.631,Z 465.355,A -85,B 0,C 180,E1 -7347.787,E2 -7347.787} C_VEL
LIN {X 0,Y 474.624,Z 465.359,A -85,B 0,C 180,E1 -7350.882,E2 -7350.882} C_VEL
LIN {X 0,Y 474.658,Z 465.346,A -85,B 0,C 180,E1 -7353.628,E2 -7353.628} C_VEL
LIN {X 0,Y 474.627,Z 465.364,A -85,B 0,C 180,E1 -7356.641,E2 -7356.641} C_VEL
LIN {X 0,Y 474.648,Z 465.353,A -85,B 0,C 180,E1 -7360.089,E2 -7360.089} C_VEL
LIN {X 0,Y 474.642,Z 465.358,A -85,B 0,C 180,E1 -7362.774,E2 -7362.774} C_VEL
LIN {X 0,Y 474.638,Z 465.358,A -85,B 0,C 180,E1 -7365.421,E2 -7365.421} C_VEL
LIN {X 0,Y 474.696,Z 465.35,A -85,B 0,C 180,E1 -7368.037,E2 -7368.037} C_VEL
LIN {X 0,Y 474.719,Z 465.347,A -85,B 0,C 180,E1 -7371.486,E2 -7371.486} C_VEL
LIN {X 0,Y 474.78,Z 465.341,A -85,B 0,C 180,E1 -7374.052,E2 -7374.052} C_VEL
LIN {X 0,Y 474.886,Z 465.325,A -85,B 0,C 180,E1 -7377.455,E2 -7377.455} C_VEL
LIN {X 0,Y 474.868,Z 465.33,A -85,B 0,C 180,E1 -7380.848,E2 -7380.848} C_VEL
LIN {X 0,Y 474.886,Z 465.326,A -85,B 0,C 180,E1 -7382.545,E2 -7382.545} C_VEL
LIN {X 0,Y 474.782,Z 465.34,A -85,B 0,C 180,E1 -7385.948,E2 -7385.948} C_VEL
